// TIA Portal V18 export
// export: Created 2025-12-01T12:38:42.0092621Z, ExportSetting None, DisplayName Totally Integrated Automation Portal, DisplayVersion V18 Update 5, DisplayName TIA Portal Openness, DisplayVersion V18 Update 5, DisplayName TIA Portal Teamcenter Gateway, DisplayVersion V18, DisplayName TIA Portal Version Control Interface, DisplayVersion V18, DisplayName STEP 7 Professional, DisplayVersion V18 Update 5, DisplayName STEP 7 Safety, DisplayVersion V18, DisplayName WinCC Professional, DisplayVersion V18 Update 5
FUNCTION "Robot" : Void   // FC2400, LAD
{ S7_Optimized_Access := 'TRUE' }
// stored: AutoNumber false, SetENOAutomatically false
   VAR_TEMP   // added for the SCL form of the ladder/FBD networks
      _w1 : Bool;
      _w2 : Bool;
      _w3 : Bool;
      _w4 : Bool;
      _w5 : Bool;
      _w6 : Bool;
   END_VAR
BEGIN

REGION Network 1: 调用机器人1 / Call robot 1
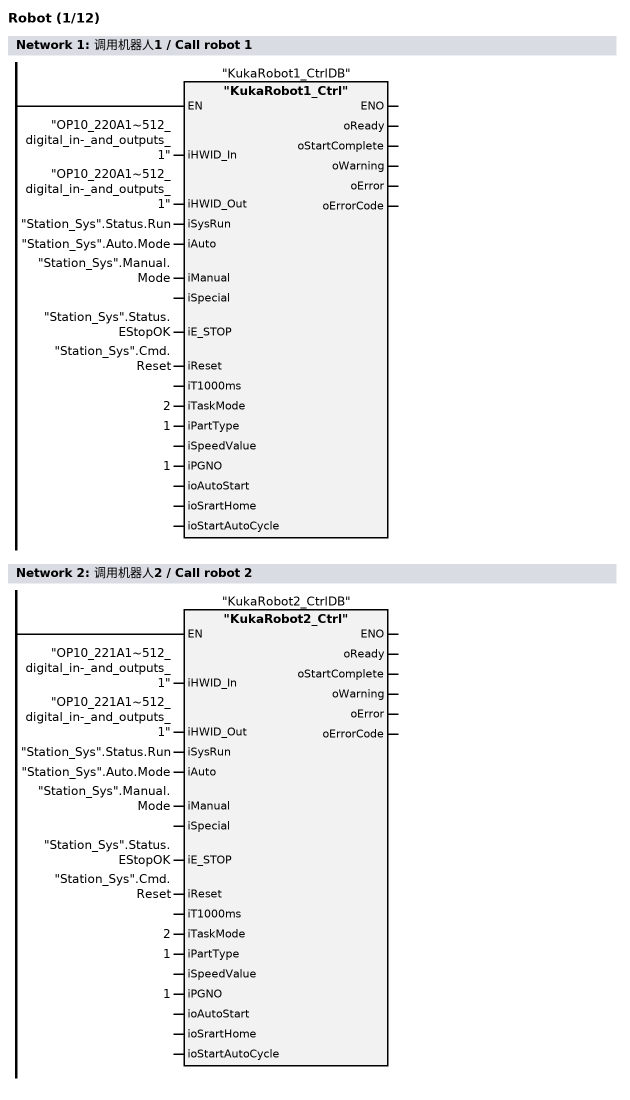
   RUNG wire#powerrail
      "KukaRobot1_CtrlDB"(iHWID_In := "OP10_220A1~512_digital_in-_and_outputs_1", iHWID_Out := "OP10_220A1~512_digital_in-_and_outputs_1", iSysRun := "Station_Sys".Status.Run, iAuto := "Station_Sys".Auto.Mode, iManual := "Station_Sys".Manual.Mode, iSpecial :=, iE_STOP := "Station_Sys".Status.EStopOK, iReset := "Station_Sys".Cmd.Reset, iT1000ms :=, iTaskMode := 2, iPartType := 1, iSpeedValue :=, iPGNO := 1, ioAutoStart :=, ioSrartHome :=, ioStartAutoCycle :=, oReady =>, oStartComplete =>, oWarning =>, oError =>, oErrorCode =>)
   END_RUNG
   // the same network as SCL:
   "KukaRobot1_CtrlDB"(iHWID_In := "OP10_220A1~512_digital_in-_and_outputs_1",   // "KukaRobot1_Ctrl"
                       iHWID_Out := "OP10_220A1~512_digital_in-_and_outputs_1",
                       iSysRun := "Station_Sys".Status.Run,
                       iAuto := "Station_Sys".Auto.Mode,
                       iManual := "Station_Sys".Manual.Mode,
                       iE_STOP := "Station_Sys".Status.EStopOK,
                       iReset := "Station_Sys".Cmd.Reset,
                       iTaskMode := 2,
                       iPartType := 1,
                       iPGNO := 1);
END_REGION

REGION Network 2: 调用机器人2 / Call robot 2
   RUNG wire#powerrail
      "KukaRobot2_CtrlDB"(iHWID_In := "OP10_221A1~512_digital_in-_and_outputs_1", iHWID_Out := "OP10_221A1~512_digital_in-_and_outputs_1", iSysRun := "Station_Sys".Status.Run, iAuto := "Station_Sys".Auto.Mode, iManual := "Station_Sys".Manual.Mode, iSpecial :=, iE_STOP := "Station_Sys".Status.EStopOK, iReset := "Station_Sys".Cmd.Reset, iT1000ms :=, iTaskMode := 2, iPartType := 1, iSpeedValue :=, iPGNO := 1, ioAutoStart :=, ioSrartHome :=, ioStartAutoCycle :=, oReady =>, oStartComplete =>, oWarning =>, oError =>, oErrorCode =>)
   END_RUNG
   // the same network as SCL:
   "KukaRobot2_CtrlDB"(iHWID_In := "OP10_221A1~512_digital_in-_and_outputs_1",   // "KukaRobot2_Ctrl"
                       iHWID_Out := "OP10_221A1~512_digital_in-_and_outputs_1",
                       iSysRun := "Station_Sys".Status.Run,
                       iAuto := "Station_Sys".Auto.Mode,
                       iManual := "Station_Sys".Manual.Mode,
                       iE_STOP := "Station_Sys".Status.EStopOK,
                       iReset := "Station_Sys".Cmd.Reset,
                       iTaskMode := 2,
                       iPartType := 1,
                       iPGNO := 1);
END_REGION

REGION Network 3: 调用机器人3 / Call robot 3
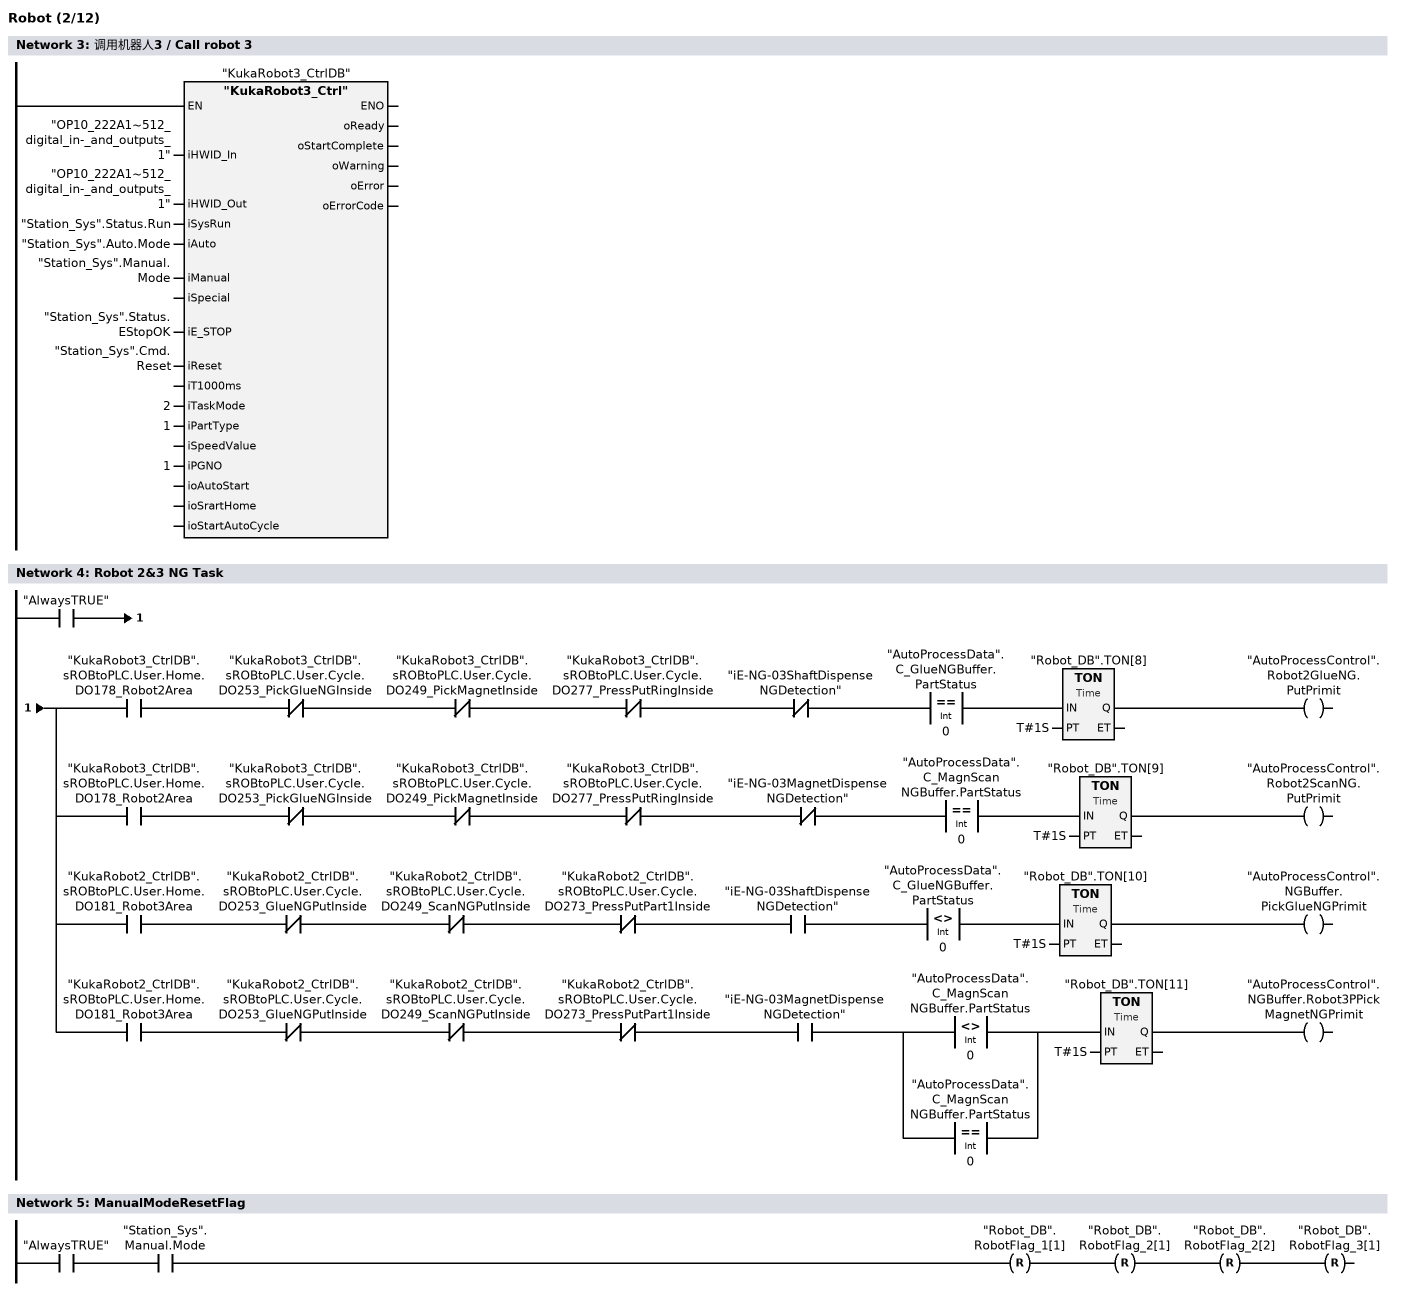
   RUNG wire#powerrail
      "KukaRobot3_CtrlDB"(iHWID_In := "OP10_222A1~512_digital_in-_and_outputs_1", iHWID_Out := "OP10_222A1~512_digital_in-_and_outputs_1", iSysRun := "Station_Sys".Status.Run, iAuto := "Station_Sys".Auto.Mode, iManual := "Station_Sys".Manual.Mode, iSpecial :=, iE_STOP := "Station_Sys".Status.EStopOK, iReset := "Station_Sys".Cmd.Reset, iT1000ms :=, iTaskMode := 2, iPartType := 1, iSpeedValue :=, iPGNO := 1, ioAutoStart :=, ioSrartHome :=, ioStartAutoCycle :=, oReady =>, oStartComplete =>, oWarning =>, oError =>, oErrorCode =>)
   END_RUNG
   // the same network as SCL:
   "KukaRobot3_CtrlDB"(iHWID_In := "OP10_222A1~512_digital_in-_and_outputs_1",   // "KukaRobot3_Ctrl"
                       iHWID_Out := "OP10_222A1~512_digital_in-_and_outputs_1",
                       iSysRun := "Station_Sys".Status.Run,
                       iAuto := "Station_Sys".Auto.Mode,
                       iManual := "Station_Sys".Manual.Mode,
                       iE_STOP := "Station_Sys".Status.EStopOK,
                       iReset := "Station_Sys".Cmd.Reset,
                       iTaskMode := 2,
                       iPartType := 1,
                       iPGNO := 1);
END_REGION

REGION Network 4: Robot 2&3 NG Task
   RUNG wire#powerrail
      Contact( "AlwaysTRUE" )
      wire#w1
      Contact( "KukaRobot3_CtrlDB".sROBtoPLC.User.Home.DO178_Robot2Area )
      I_Contact( "KukaRobot3_CtrlDB".sROBtoPLC.User.Cycle.DO253_PickGlueNGInside )
      I_Contact( "KukaRobot3_CtrlDB".sROBtoPLC.User.Cycle.DO249_PickMagnetInside )
      I_Contact( "KukaRobot3_CtrlDB".sROBtoPLC.User.Cycle.DO277_PressPutRingInside )
      I_Contact( "iE-NG-03ShaftDispenseNGDetection" )
      { S7_Templates := "SrcType := Int" } EQ_Contact(in1 := "AutoProcessData".C_GlueNGBuffer.PartStatus, in2 := 0)
      { S7_Templates := "time_type := Time" } "Robot_DB".TON[8].TON(pt := T#1S, et =>)
      Coil( "AutoProcessControl".Robot2GlueNG.PutPrimit )
   END_RUNG
   RUNG wire#w1
      Contact( "KukaRobot3_CtrlDB".sROBtoPLC.User.Home.DO178_Robot2Area )
      I_Contact( "KukaRobot3_CtrlDB".sROBtoPLC.User.Cycle.DO253_PickGlueNGInside )
      I_Contact( "KukaRobot3_CtrlDB".sROBtoPLC.User.Cycle.DO249_PickMagnetInside )
      I_Contact( "KukaRobot3_CtrlDB".sROBtoPLC.User.Cycle.DO277_PressPutRingInside )
      I_Contact( "iE-NG-03MagnetDispenseNGDetection" )
      { S7_Templates := "SrcType := Int" } EQ_Contact(in1 := "AutoProcessData".C_MagnScanNGBuffer.PartStatus, in2 := 0)
      { S7_Templates := "time_type := Time" } "Robot_DB".TON[9].TON(pt := T#1S, et =>)
      Coil( "AutoProcessControl".Robot2ScanNG.PutPrimit )
   END_RUNG
   RUNG wire#w1
      Contact( "KukaRobot2_CtrlDB".sROBtoPLC.User.Home.DO181_Robot3Area )
      I_Contact( "KukaRobot2_CtrlDB".sROBtoPLC.User.Cycle.DO253_GlueNGPutInside )
      I_Contact( "KukaRobot2_CtrlDB".sROBtoPLC.User.Cycle.DO249_ScanNGPutInside )
      I_Contact( "KukaRobot2_CtrlDB".sROBtoPLC.User.Cycle.DO273_PressPutPart1Inside )
      Contact( "iE-NG-03ShaftDispenseNGDetection" )
      { S7_Templates := "SrcType := Int" } NE_Contact(in1 := "AutoProcessData".C_GlueNGBuffer.PartStatus, in2 := 0)
      { S7_Templates := "time_type := Time" } "Robot_DB".TON[10].TON(pt := T#1S, et =>)
      Coil( "AutoProcessControl".NGBuffer.PickGlueNGPrimit )
   END_RUNG
   RUNG wire#w1
      Contact( "KukaRobot2_CtrlDB".sROBtoPLC.User.Home.DO181_Robot3Area )
      I_Contact( "KukaRobot2_CtrlDB".sROBtoPLC.User.Cycle.DO253_GlueNGPutInside )
      I_Contact( "KukaRobot2_CtrlDB".sROBtoPLC.User.Cycle.DO249_ScanNGPutInside )
      I_Contact( "KukaRobot2_CtrlDB".sROBtoPLC.User.Cycle.DO273_PressPutPart1Inside )
      Contact( "iE-NG-03MagnetDispenseNGDetection" )
      wire#w2
      { S7_Templates := "SrcType := Int" } NE_Contact(in1 := "AutoProcessData".C_MagnScanNGBuffer.PartStatus, in2 := 0)
      wire#w3
      { S7_Templates := "time_type := Time" } "Robot_DB".TON[11].TON(pt := T#1S, et =>)
      Coil( "AutoProcessControl".NGBuffer.Robot3PPickMagnetNGPrimit )
   END_RUNG
   RUNG wire#w2
      { S7_Templates := "SrcType := Int" } EQ_Contact(in1 := "AutoProcessData".C_MagnScanNGBuffer.PartStatus, in2 := 0)
   END_RUNG wire#w3
   // the same network as SCL:
   "Robot_DB".TON[8].TON(IN := "AlwaysTRUE" AND "KukaRobot3_CtrlDB".sROBtoPLC.User.Home.DO178_Robot2Area AND NOT "KukaRobot3_CtrlDB".sROBtoPLC.User.Cycle.DO253_PickGlueNGInside AND NOT "KukaRobot3_CtrlDB".sROBtoPLC.User.Cycle.DO249_PickMagnetInside AND NOT "KukaRobot3_CtrlDB".sROBtoPLC.User.Cycle.DO277_PressPutRingInside AND NOT "iE-NG-03ShaftDispenseNGDetection" AND ("AutoProcessData".C_GlueNGBuffer.PartStatus = 0),
                         PT := T#1S);
   "AutoProcessControl".Robot2GlueNG.PutPrimit := "Robot_DB".TON[8].Q;
   "Robot_DB".TON[9].TON(IN := "AlwaysTRUE" AND "KukaRobot3_CtrlDB".sROBtoPLC.User.Home.DO178_Robot2Area AND NOT "KukaRobot3_CtrlDB".sROBtoPLC.User.Cycle.DO253_PickGlueNGInside AND NOT "KukaRobot3_CtrlDB".sROBtoPLC.User.Cycle.DO249_PickMagnetInside AND NOT "KukaRobot3_CtrlDB".sROBtoPLC.User.Cycle.DO277_PressPutRingInside AND NOT "iE-NG-03MagnetDispenseNGDetection" AND ("AutoProcessData".C_MagnScanNGBuffer.PartStatus = 0),
                         PT := T#1S);
   "AutoProcessControl".Robot2ScanNG.PutPrimit := "Robot_DB".TON[9].Q;
   "Robot_DB".TON[10].TON(IN := "AlwaysTRUE" AND "KukaRobot2_CtrlDB".sROBtoPLC.User.Home.DO181_Robot3Area AND NOT "KukaRobot2_CtrlDB".sROBtoPLC.User.Cycle.DO253_GlueNGPutInside AND NOT "KukaRobot2_CtrlDB".sROBtoPLC.User.Cycle.DO249_ScanNGPutInside AND NOT "KukaRobot2_CtrlDB".sROBtoPLC.User.Cycle.DO273_PressPutPart1Inside AND "iE-NG-03ShaftDispenseNGDetection" AND ("AutoProcessData".C_GlueNGBuffer.PartStatus <> 0),
                          PT := T#1S);
   "AutoProcessControl".NGBuffer.PickGlueNGPrimit := "Robot_DB".TON[10].Q;
   "Robot_DB".TON[11].TON(IN := "AlwaysTRUE" AND "KukaRobot2_CtrlDB".sROBtoPLC.User.Home.DO181_Robot3Area AND NOT "KukaRobot2_CtrlDB".sROBtoPLC.User.Cycle.DO253_GlueNGPutInside AND NOT "KukaRobot2_CtrlDB".sROBtoPLC.User.Cycle.DO249_ScanNGPutInside AND NOT "KukaRobot2_CtrlDB".sROBtoPLC.User.Cycle.DO273_PressPutPart1Inside AND "iE-NG-03MagnetDispenseNGDetection" AND (("AutoProcessData".C_MagnScanNGBuffer.PartStatus <> 0) OR ("AutoProcessData".C_MagnScanNGBuffer.PartStatus = 0)),
                          PT := T#1S);
   "AutoProcessControl".NGBuffer.Robot3PPickMagnetNGPrimit := "Robot_DB".TON[11].Q;
END_REGION

REGION Network 5: ManualModeResetFlag
   RUNG wire#powerrail
      Contact( "AlwaysTRUE" )
      Contact( "Station_Sys".Manual.Mode )
      R_Coil( "Robot_DB".RobotFlag_1[1] )
      R_Coil( "Robot_DB".RobotFlag_2[1] )
      R_Coil( "Robot_DB".RobotFlag_2[2] )
      R_Coil( "Robot_DB".RobotFlag_3[1] )
   END_RUNG
   // the same network as SCL:
   IF "AlwaysTRUE" AND "Station_Sys".Manual.Mode THEN
       "Robot_DB".RobotFlag_1[1] := FALSE;
       "Robot_DB".RobotFlag_2[1] := FALSE;
       "Robot_DB".RobotFlag_2[2] := FALSE;
       "Robot_DB".RobotFlag_3[1] := FALSE;
   END_IF;
END_REGION

REGION Network 6 (SCL): LoadNG传感器 / Loadng sensor
   //NG1
   "KukaRobot1_CtrlDB".sPLCtoROB.User.Home.DI177_NG1_1:="Robot_DB".LoadNG_1[1] := "iE1-UnloadingShaftPressNG_5";
   "KukaRobot1_CtrlDB".sPLCtoROB.User.Home.DI178_NG1_2:="Robot_DB".LoadNG_1[2] := "iE1-UnloadingShaftPressNG_4";
   "KukaRobot1_CtrlDB".sPLCtoROB.User.Home.DI179_NG1_3:="Robot_DB".LoadNG_1[3] := "iE1-UnloadingShaftPressNG_3";
   "KukaRobot1_CtrlDB".sPLCtoROB.User.Home.DI180_NG1_4:="Robot_DB".LoadNG_1[4] := "iE1-UnloadingShaftPressNG_2";
   "KukaRobot1_CtrlDB".sPLCtoROB.User.Home.DI181_NG1_5:="Robot_DB".LoadNG_1[5] := "iE1-UnloadingShaftPressNG_1";

   //NG2
   "KukaRobot1_CtrlDB".sPLCtoROB.User.Home.DI182_NG2_1:="Robot_DB".LoadNG_2[1] := "iE1-UnloadingShaftScanNG_5";
   "KukaRobot1_CtrlDB".sPLCtoROB.User.Home.DI183_NG2_2:="Robot_DB".LoadNG_2[2] := "iE1-UnloadingShaftScanNG_4";
   "KukaRobot1_CtrlDB".sPLCtoROB.User.Home.DI184_NG2_3:="Robot_DB".LoadNG_2[3] := "iE1-UnloadingShaftScanNG_3";
   "KukaRobot1_CtrlDB".sPLCtoROB.User.Home.DI185_NG2_4:="Robot_DB".LoadNG_2[4] := "iE1-UnloadingShaftScanNG_2";
   "KukaRobot1_CtrlDB".sPLCtoROB.User.Home.DI186_NG2_5:="Robot_DB".LoadNG_2[5] := "iE1-UnloadingShaftScanNG_1";

   //NG3
   "KukaRobot1_CtrlDB".sPLCtoROB.User.Home.DI187_NG3_1:="Robot_DB".LoadNG_3[1] := "iE1-UnloadingRingScanNG_5";
   "KukaRobot1_CtrlDB".sPLCtoROB.User.Home.DI188_NG3_2:="Robot_DB".LoadNG_3[2] := "iE1-UnloadingRingScanNG_4";
   "KukaRobot1_CtrlDB".sPLCtoROB.User.Home.DI189_NG3_3:="Robot_DB".LoadNG_3[3] := "iE1-UnloadingRingScanNG_3";
   "KukaRobot1_CtrlDB".sPLCtoROB.User.Home.DI190_NG3_4:="Robot_DB".LoadNG_3[4] := "iE1-UnloadingRingScanNG_2";
   "KukaRobot1_CtrlDB".sPLCtoROB.User.Home.DI191_NG3_5:="Robot_DB".LoadNG_3[5] := "iE1-UnloadingRingScanNG_1";
END_REGION

REGION Network 7 (SCL): UnLoadNG传感器 / UnLoadNG sensor
   //NG1
   "KukaRobot3_CtrlDB".sPLCtoROB.User.Home.DI177_PressNG1_1:="Robot_DB".UnLoadNG_1[1] := "iE2-UnloadingPressNG_5";
   "KukaRobot3_CtrlDB".sPLCtoROB.User.Home.DI178_PressNG1_2:="Robot_DB".UnLoadNG_1[2] := "iE2-UnloadingPressNG_4";
   "KukaRobot3_CtrlDB".sPLCtoROB.User.Home.DI179_PressNG1_3:="Robot_DB".UnLoadNG_1[3] := "iE2-UnloadingPressNG_3";
   "KukaRobot3_CtrlDB".sPLCtoROB.User.Home.DI180_PressNG1_4:="Robot_DB".UnLoadNG_1[4] := "iE2-UnloadingPressNG_2";
   "KukaRobot3_CtrlDB".sPLCtoROB.User.Home.DI181_PressNG1_5:="Robot_DB".UnLoadNG_1[5] := "iE2-UnloadingPressNG_1";

   //NG2
   "KukaRobot3_CtrlDB".sPLCtoROB.User.Home.DI182_GlueNG2_1:="Robot_DB".UnLoadNG_2[1] := "iE2-UnloadingMagentScanNG_5";
   "KukaRobot3_CtrlDB".sPLCtoROB.User.Home.DI183_GlueNG2_2:="Robot_DB".UnLoadNG_2[2] := "iE2-UnloadingMagentScanNG_4";
   "KukaRobot3_CtrlDB".sPLCtoROB.User.Home.DI184_GlueNG2_3:="Robot_DB".UnLoadNG_2[3] := "iE2-UnloadingMagentScanNG_3";
   "KukaRobot3_CtrlDB".sPLCtoROB.User.Home.DI185_GlueNG2_4:="Robot_DB".UnLoadNG_2[4] := "iE2-UnloadingMagentScanNG_2";
   "KukaRobot3_CtrlDB".sPLCtoROB.User.Home.DI186_GlueNG2_5:="Robot_DB".UnLoadNG_2[5] := "iE2-UnloadingMagentScanNG_1";

   //NG3
   "KukaRobot3_CtrlDB".sPLCtoROB.User.Home.DI187_ScanNG3_1:="Robot_DB".UnLoadNG_3[1] := "iE2-UnloadingRingScanNG_5";
   "KukaRobot3_CtrlDB".sPLCtoROB.User.Home.DI188_ScanNG3_2:="Robot_DB".UnLoadNG_3[2] := "iE2-UnloadingRingScanNG_4";
   "KukaRobot3_CtrlDB".sPLCtoROB.User.Home.DI189_ScanNG3_3:="Robot_DB".UnLoadNG_3[3] := "iE2-UnloadingRingScanNG_3";
   "KukaRobot3_CtrlDB".sPLCtoROB.User.Home.DI190_ScanNG3_4:="Robot_DB".UnLoadNG_3[4] := "iE2-UnloadingRingScanNG_2";
   "KukaRobot3_CtrlDB".sPLCtoROB.User.Home.DI191_ScanNG3_5:="Robot_DB".UnLoadNG_3[5] := "iE2-UnloadingRingScanNG_1";
END_REGION

REGION Network 8: RobotGripControl
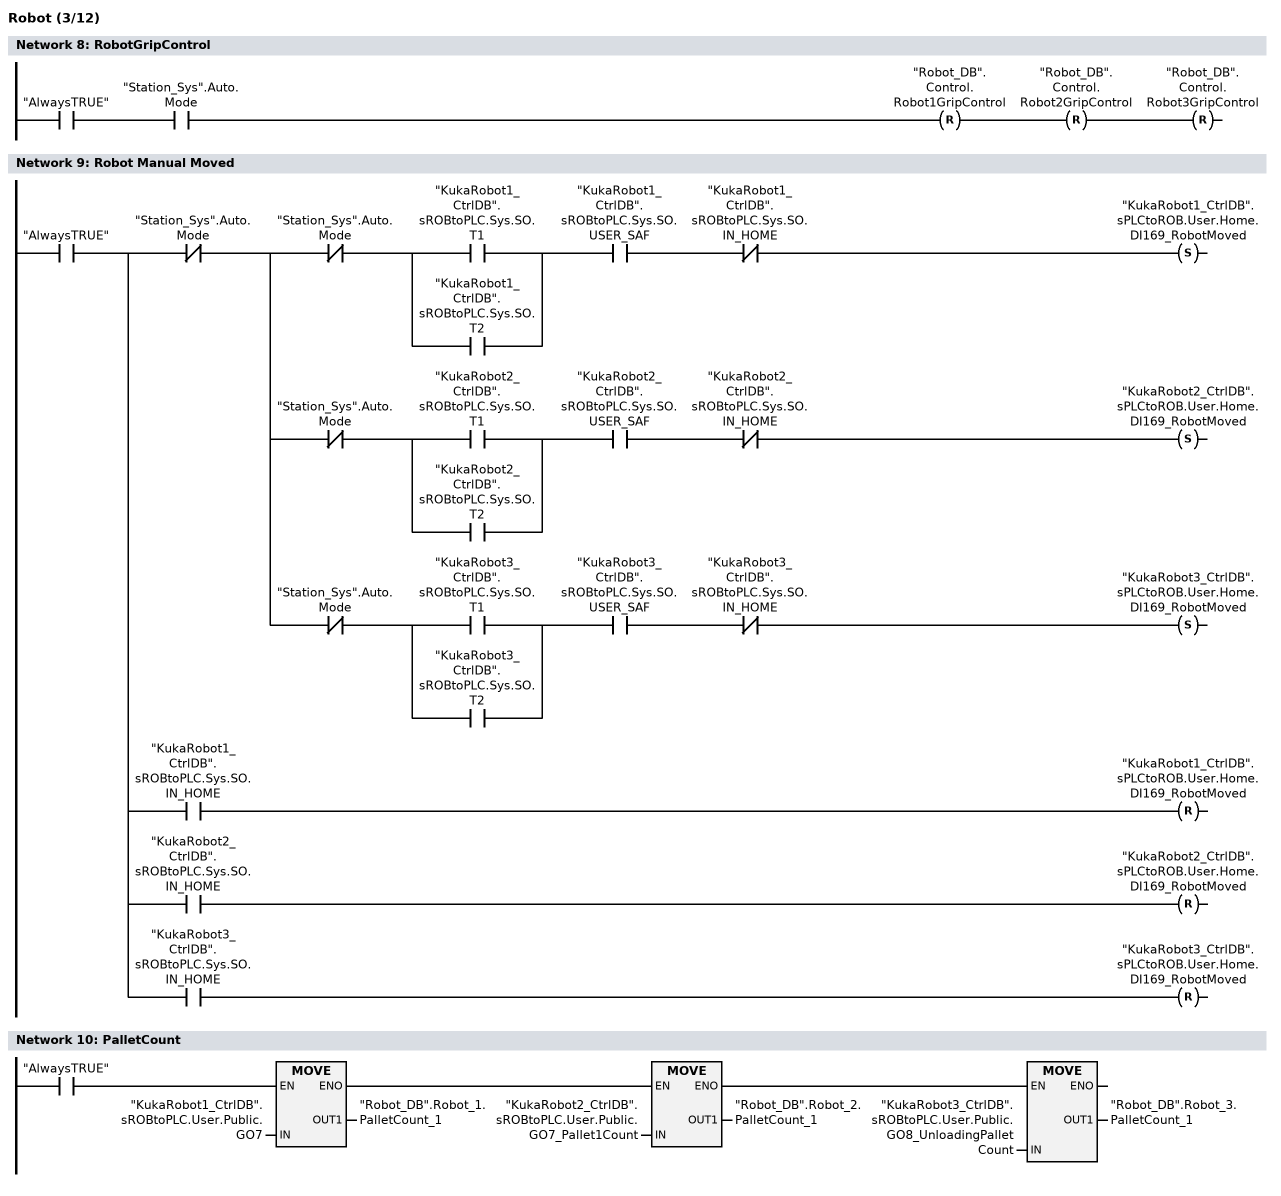
   RUNG wire#powerrail
      Contact( "AlwaysTRUE" )
      Contact( "Station_Sys".Auto.Mode )
      R_Coil( "Robot_DB".Control.Robot1GripControl )
      R_Coil( "Robot_DB".Control.Robot2GripControl )
      R_Coil( "Robot_DB".Control.Robot3GripControl )
   END_RUNG
   // the same network as SCL:
   IF "AlwaysTRUE" AND "Station_Sys".Auto.Mode THEN
       "Robot_DB".Control.Robot1GripControl := FALSE;
       "Robot_DB".Control.Robot2GripControl := FALSE;
       "Robot_DB".Control.Robot3GripControl := FALSE;
   END_IF;
END_REGION

REGION Network 9: Robot Manual Moved
   RUNG wire#powerrail
      Contact( "AlwaysTRUE" )
      wire#w1
      I_Contact( "Station_Sys".Auto.Mode )
      wire#w2
      I_Contact( "Station_Sys".Auto.Mode )
      wire#w3
      Contact( "KukaRobot1_CtrlDB".sROBtoPLC.Sys.SO.T1 )
      wire#w4
      Contact( "KukaRobot1_CtrlDB".sROBtoPLC.Sys.SO.USER_SAF )
      I_Contact( "KukaRobot1_CtrlDB".sROBtoPLC.Sys.SO.IN_HOME )
      S_Coil( "KukaRobot1_CtrlDB".sPLCtoROB.User.Home.DI169_RobotMoved )
   END_RUNG
   RUNG wire#w3
      Contact( "KukaRobot1_CtrlDB".sROBtoPLC.Sys.SO.T2 )
   END_RUNG wire#w4
   RUNG wire#w2
      I_Contact( "Station_Sys".Auto.Mode )
      wire#w5
      Contact( "KukaRobot2_CtrlDB".sROBtoPLC.Sys.SO.T1 )
      wire#w6
      Contact( "KukaRobot2_CtrlDB".sROBtoPLC.Sys.SO.USER_SAF )
      I_Contact( "KukaRobot2_CtrlDB".sROBtoPLC.Sys.SO.IN_HOME )
      S_Coil( "KukaRobot2_CtrlDB".sPLCtoROB.User.Home.DI169_RobotMoved )
   END_RUNG
   RUNG wire#w5
      Contact( "KukaRobot2_CtrlDB".sROBtoPLC.Sys.SO.T2 )
   END_RUNG wire#w6
   RUNG wire#w2
      I_Contact( "Station_Sys".Auto.Mode )
      wire#w7
      Contact( "KukaRobot3_CtrlDB".sROBtoPLC.Sys.SO.T1 )
      wire#w8
      Contact( "KukaRobot3_CtrlDB".sROBtoPLC.Sys.SO.USER_SAF )
      I_Contact( "KukaRobot3_CtrlDB".sROBtoPLC.Sys.SO.IN_HOME )
      S_Coil( "KukaRobot3_CtrlDB".sPLCtoROB.User.Home.DI169_RobotMoved )
   END_RUNG
   RUNG wire#w7
      Contact( "KukaRobot3_CtrlDB".sROBtoPLC.Sys.SO.T2 )
   END_RUNG wire#w8
   RUNG wire#w1
      Contact( "KukaRobot1_CtrlDB".sROBtoPLC.Sys.SO.IN_HOME )
      R_Coil( "KukaRobot1_CtrlDB".sPLCtoROB.User.Home.DI169_RobotMoved )
   END_RUNG
   RUNG wire#w1
      Contact( "KukaRobot2_CtrlDB".sROBtoPLC.Sys.SO.IN_HOME )
      R_Coil( "KukaRobot2_CtrlDB".sPLCtoROB.User.Home.DI169_RobotMoved )
   END_RUNG
   RUNG wire#w1
      Contact( "KukaRobot3_CtrlDB".sROBtoPLC.Sys.SO.IN_HOME )
      R_Coil( "KukaRobot3_CtrlDB".sPLCtoROB.User.Home.DI169_RobotMoved )
   END_RUNG
   // the same network as SCL:
   #_w1 := "AlwaysTRUE" AND NOT "Station_Sys".Auto.Mode;
   IF #_w1 AND NOT "Station_Sys".Auto.Mode AND ("KukaRobot1_CtrlDB".sROBtoPLC.Sys.SO.T1 OR "KukaRobot1_CtrlDB".sROBtoPLC.Sys.SO.T2) AND "KukaRobot1_CtrlDB".sROBtoPLC.Sys.SO.USER_SAF AND NOT "KukaRobot1_CtrlDB".sROBtoPLC.Sys.SO.IN_HOME THEN
       "KukaRobot1_CtrlDB".sPLCtoROB.User.Home.DI169_RobotMoved := TRUE;
   END_IF;
   IF #_w1 AND NOT "Station_Sys".Auto.Mode AND ("KukaRobot2_CtrlDB".sROBtoPLC.Sys.SO.T1 OR "KukaRobot2_CtrlDB".sROBtoPLC.Sys.SO.T2) AND "KukaRobot2_CtrlDB".sROBtoPLC.Sys.SO.USER_SAF AND NOT "KukaRobot2_CtrlDB".sROBtoPLC.Sys.SO.IN_HOME THEN
       "KukaRobot2_CtrlDB".sPLCtoROB.User.Home.DI169_RobotMoved := TRUE;
   END_IF;
   IF #_w1 AND NOT "Station_Sys".Auto.Mode AND ("KukaRobot3_CtrlDB".sROBtoPLC.Sys.SO.T1 OR "KukaRobot3_CtrlDB".sROBtoPLC.Sys.SO.T2) AND "KukaRobot3_CtrlDB".sROBtoPLC.Sys.SO.USER_SAF AND NOT "KukaRobot3_CtrlDB".sROBtoPLC.Sys.SO.IN_HOME THEN
       "KukaRobot3_CtrlDB".sPLCtoROB.User.Home.DI169_RobotMoved := TRUE;
   END_IF;
   IF "AlwaysTRUE" AND "KukaRobot1_CtrlDB".sROBtoPLC.Sys.SO.IN_HOME THEN
       "KukaRobot1_CtrlDB".sPLCtoROB.User.Home.DI169_RobotMoved := FALSE;
   END_IF;
   IF "AlwaysTRUE" AND "KukaRobot2_CtrlDB".sROBtoPLC.Sys.SO.IN_HOME THEN
       "KukaRobot2_CtrlDB".sPLCtoROB.User.Home.DI169_RobotMoved := FALSE;
   END_IF;
   IF "AlwaysTRUE" AND "KukaRobot3_CtrlDB".sROBtoPLC.Sys.SO.IN_HOME THEN
       "KukaRobot3_CtrlDB".sPLCtoROB.User.Home.DI169_RobotMoved := FALSE;
   END_IF;
END_REGION

REGION Network 10: PalletCount
   RUNG wire#powerrail
      Contact( "AlwaysTRUE" )
      Move(in := "KukaRobot1_CtrlDB".sROBtoPLC.User.Public.GO7, out1 => "Robot_DB".Robot_1.PalletCount_1)
      Move(in := "KukaRobot2_CtrlDB".sROBtoPLC.User.Public.GO7_Pallet1Count, out1 => "Robot_DB".Robot_2.PalletCount_1)
      Move(in := "KukaRobot3_CtrlDB".sROBtoPLC.User.Public.GO8_UnloadingPalletCount, out1 => "Robot_DB".Robot_3.PalletCount_1)
   END_RUNG
   // the same network as SCL:
   IF "AlwaysTRUE" THEN
       "Robot_DB".Robot_1.PalletCount_1 := "KukaRobot1_CtrlDB".sROBtoPLC.User.Public.GO7;
       "Robot_DB".Robot_2.PalletCount_1 := "KukaRobot2_CtrlDB".sROBtoPLC.User.Public.GO7_Pallet1Count;
       "Robot_DB".Robot_3.PalletCount_1 := "KukaRobot3_CtrlDB".sROBtoPLC.User.Public.GO8_UnloadingPalletCount;
   END_IF;
END_REGION

REGION Network 12: ----------------------------------------- Robot_1 -------------------------------------
END_REGION

REGION Network 13: CodeCompare
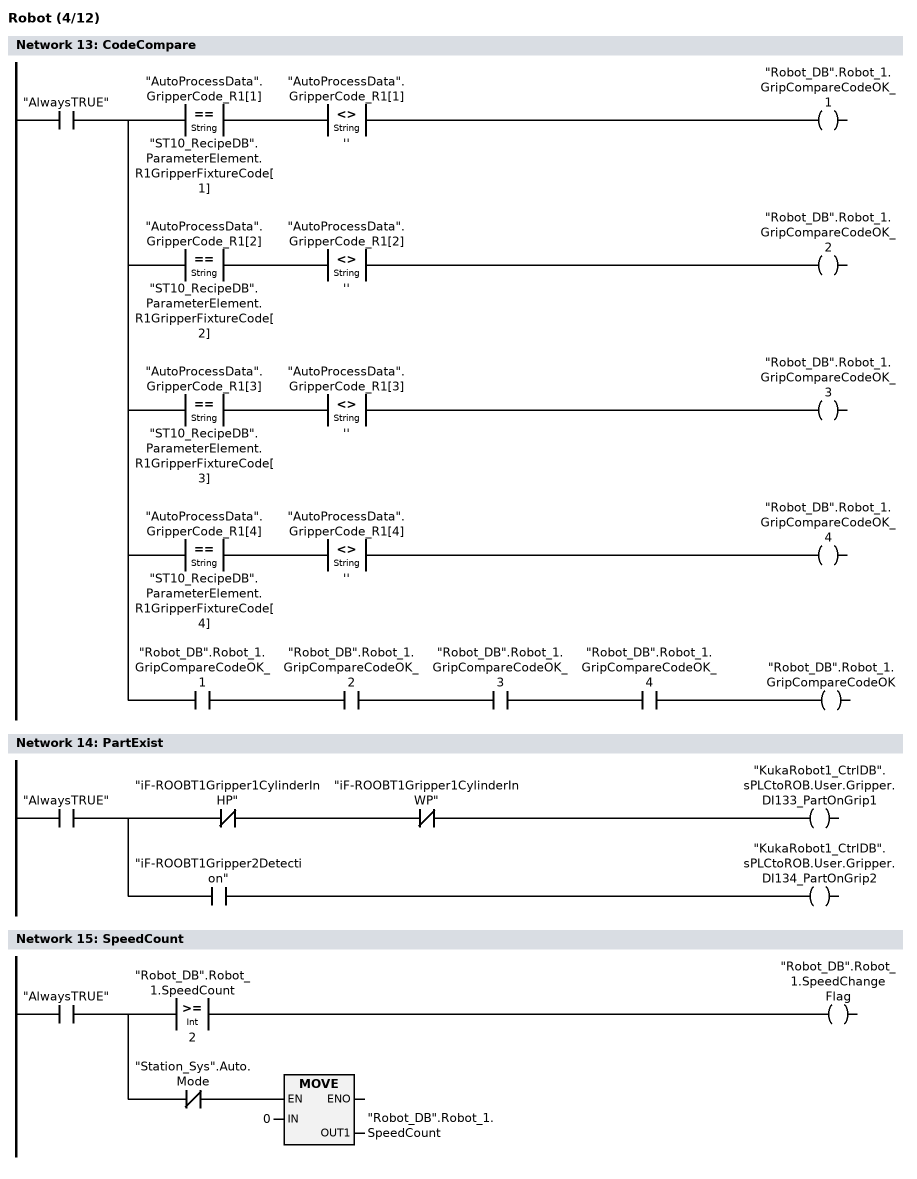
   RUNG wire#powerrail
      Contact( "AlwaysTRUE" )
      wire#w1
      { S7_Templates := "SrcType := String" } EQ_Contact(in1 := "AutoProcessData".GripperCode_R1[1], in2 := "ST10_RecipeDB".ParameterElement.R1GripperFixtureCode[1])
      { S7_Templates := "SrcType := String" } NE_Contact(in1 := "AutoProcessData".GripperCode_R1[1], in2 := '')
      Coil( "Robot_DB".Robot_1.GripCompareCodeOK_1 )
   END_RUNG
   RUNG wire#w1
      { S7_Templates := "SrcType := String" } EQ_Contact(in1 := "AutoProcessData".GripperCode_R1[2], in2 := "ST10_RecipeDB".ParameterElement.R1GripperFixtureCode[2])
      { S7_Templates := "SrcType := String" } NE_Contact(in1 := "AutoProcessData".GripperCode_R1[2], in2 := '')
      Coil( "Robot_DB".Robot_1.GripCompareCodeOK_2 )
   END_RUNG
   RUNG wire#w1
      { S7_Templates := "SrcType := String" } EQ_Contact(in1 := "AutoProcessData".GripperCode_R1[3], in2 := "ST10_RecipeDB".ParameterElement.R1GripperFixtureCode[3])
      { S7_Templates := "SrcType := String" } NE_Contact(in1 := "AutoProcessData".GripperCode_R1[3], in2 := '')
      Coil( "Robot_DB".Robot_1.GripCompareCodeOK_3 )
   END_RUNG
   RUNG wire#w1
      { S7_Templates := "SrcType := String" } EQ_Contact(in1 := "AutoProcessData".GripperCode_R1[4], in2 := "ST10_RecipeDB".ParameterElement.R1GripperFixtureCode[4])
      { S7_Templates := "SrcType := String" } NE_Contact(in1 := "AutoProcessData".GripperCode_R1[4], in2 := '')
      Coil( "Robot_DB".Robot_1.GripCompareCodeOK_4 )
   END_RUNG
   RUNG wire#w1
      Contact( "Robot_DB".Robot_1.GripCompareCodeOK_1 )
      Contact( "Robot_DB".Robot_1.GripCompareCodeOK_2 )
      Contact( "Robot_DB".Robot_1.GripCompareCodeOK_3 )
      Contact( "Robot_DB".Robot_1.GripCompareCodeOK_4 )
      Coil( "Robot_DB".Robot_1.GripCompareCodeOK )
   END_RUNG
   // the same network as SCL:
   "Robot_DB".Robot_1.GripCompareCodeOK_1 := "AlwaysTRUE" AND ("AutoProcessData".GripperCode_R1[1] = "ST10_RecipeDB".ParameterElement.R1GripperFixtureCode[1]) AND ("AutoProcessData".GripperCode_R1[1] <> '');
   "Robot_DB".Robot_1.GripCompareCodeOK_2 := "AlwaysTRUE" AND ("AutoProcessData".GripperCode_R1[2] = "ST10_RecipeDB".ParameterElement.R1GripperFixtureCode[2]) AND ("AutoProcessData".GripperCode_R1[2] <> '');
   "Robot_DB".Robot_1.GripCompareCodeOK_3 := "AlwaysTRUE" AND ("AutoProcessData".GripperCode_R1[3] = "ST10_RecipeDB".ParameterElement.R1GripperFixtureCode[3]) AND ("AutoProcessData".GripperCode_R1[3] <> '');
   "Robot_DB".Robot_1.GripCompareCodeOK_4 := "AlwaysTRUE" AND ("AutoProcessData".GripperCode_R1[4] = "ST10_RecipeDB".ParameterElement.R1GripperFixtureCode[4]) AND ("AutoProcessData".GripperCode_R1[4] <> '');
   "Robot_DB".Robot_1.GripCompareCodeOK := "AlwaysTRUE" AND "Robot_DB".Robot_1.GripCompareCodeOK_1 AND "Robot_DB".Robot_1.GripCompareCodeOK_2 AND "Robot_DB".Robot_1.GripCompareCodeOK_3 AND "Robot_DB".Robot_1.GripCompareCodeOK_4;
END_REGION

REGION Network 14: PartExist
   RUNG wire#powerrail
      Contact( "AlwaysTRUE" )
      wire#w1
      I_Contact( "iF-ROOBT1Gripper1CylinderInHP" )
      I_Contact( "iF-ROOBT1Gripper1CylinderInWP" )
      Coil( "KukaRobot1_CtrlDB".sPLCtoROB.User.Gripper.DI133_PartOnGrip1 )
   END_RUNG
   RUNG wire#w1
      Contact( "iF-ROOBT1Gripper2Detection" )
      Coil( "KukaRobot1_CtrlDB".sPLCtoROB.User.Gripper.DI134_PartOnGrip2 )
   END_RUNG
   // the same network as SCL:
   "KukaRobot1_CtrlDB".sPLCtoROB.User.Gripper.DI133_PartOnGrip1 := "AlwaysTRUE" AND NOT "iF-ROOBT1Gripper1CylinderInHP" AND NOT "iF-ROOBT1Gripper1CylinderInWP";
   "KukaRobot1_CtrlDB".sPLCtoROB.User.Gripper.DI134_PartOnGrip2 := "AlwaysTRUE" AND "iF-ROOBT1Gripper2Detection";
END_REGION

REGION Network 15: SpeedCount
   RUNG wire#powerrail
      Contact( "AlwaysTRUE" )
      wire#w1
      { S7_Templates := "SrcType := Int" } GE_Contact(in1 := "Robot_DB".Robot_1.SpeedCount, in2 := 2)
      Coil( "Robot_DB".Robot_1.SpeedChangeFlag )
   END_RUNG
   RUNG wire#w1
      I_Contact( "Station_Sys".Auto.Mode )
      Move(in := 0, out1 => "Robot_DB".Robot_1.SpeedCount)
   END_RUNG
   // the same network as SCL:
   "Robot_DB".Robot_1.SpeedChangeFlag := "AlwaysTRUE" AND ("Robot_DB".Robot_1.SpeedCount >= 2);
   IF "AlwaysTRUE" AND NOT "Station_Sys".Auto.Mode THEN "Robot_DB".Robot_1.SpeedCount := 0; END_IF;
END_REGION

REGION Network 16: Robot1Speed Interlock
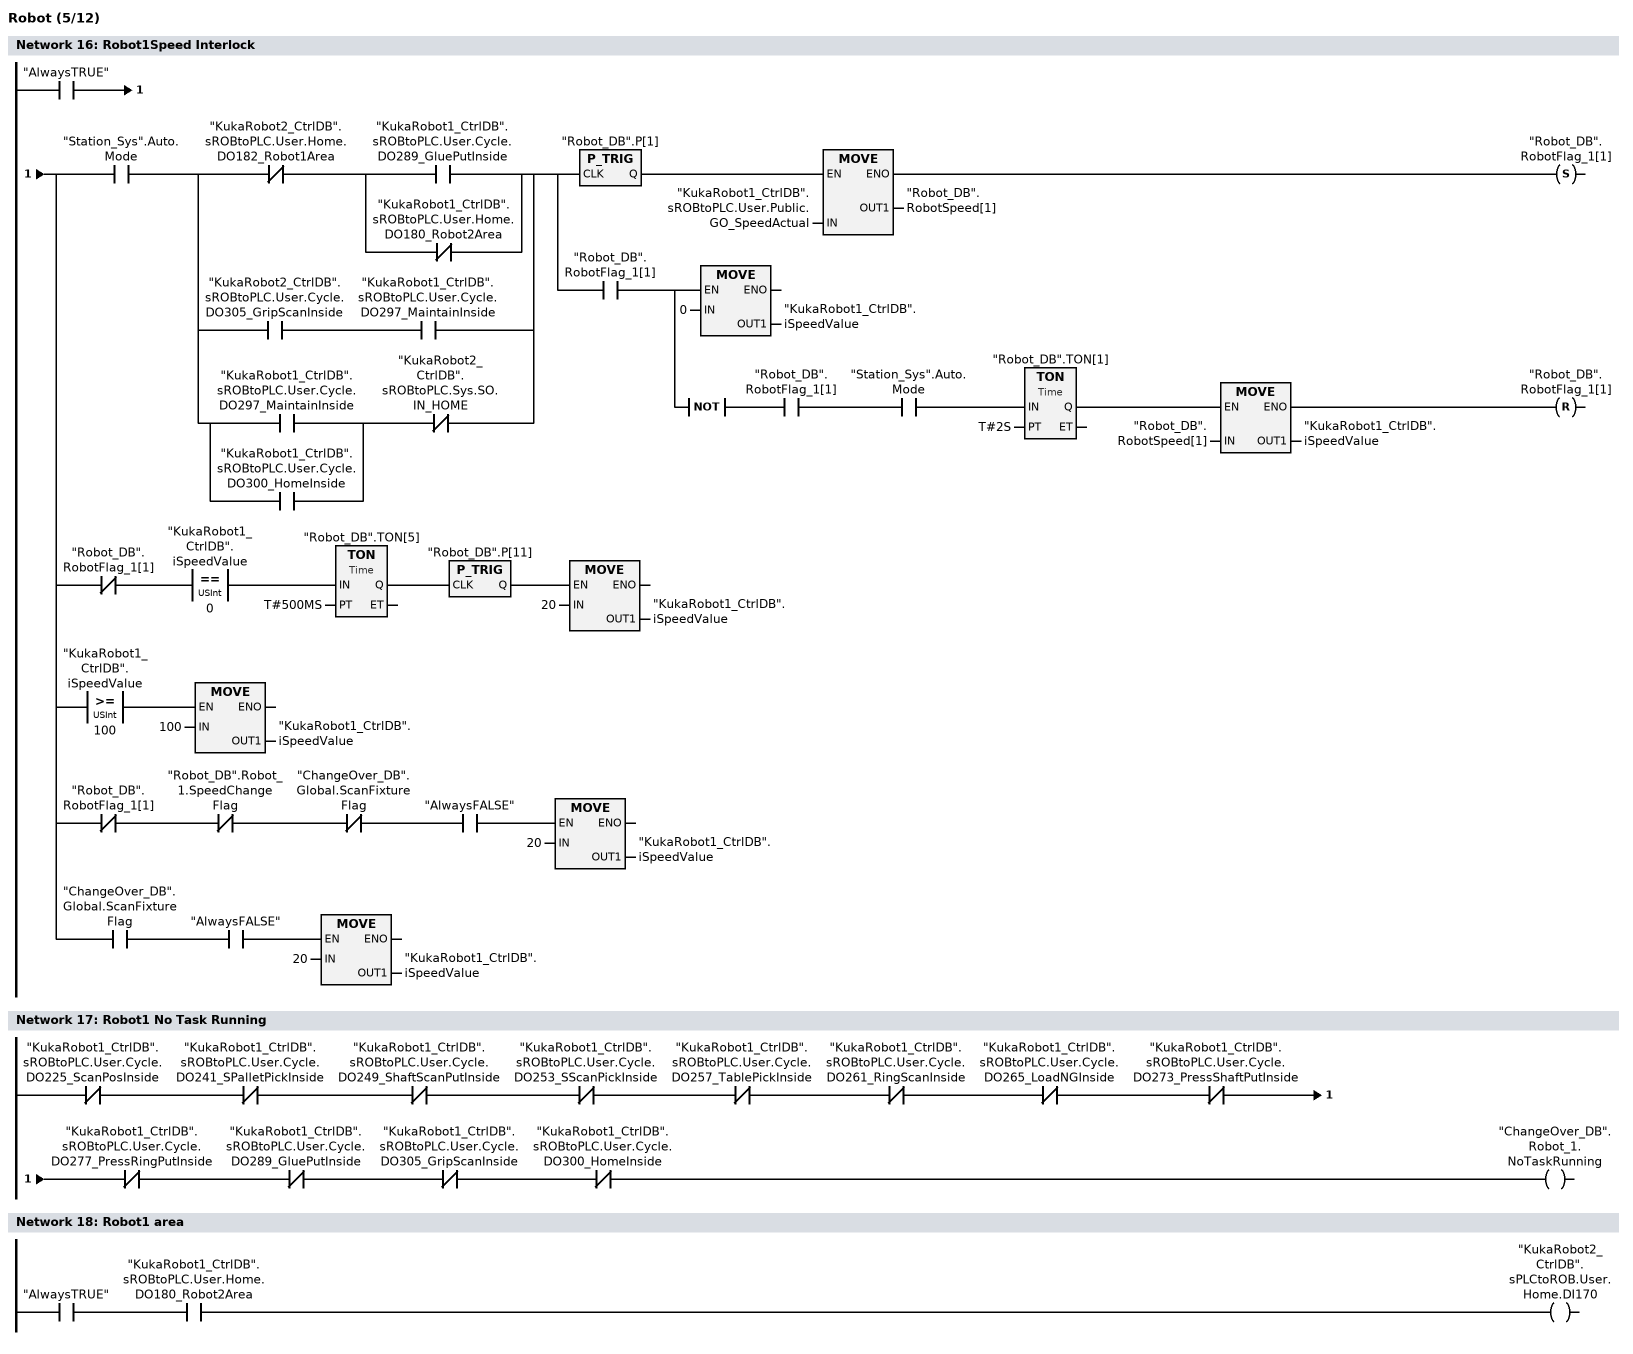
   RUNG wire#powerrail
      Contact( "AlwaysTRUE" )
      wire#w1
      Contact( "Station_Sys".Auto.Mode )
      wire#w2
      I_Contact( "KukaRobot2_CtrlDB".sROBtoPLC.User.Home.DO182_Robot1Area )
      wire#w3
      Contact( "KukaRobot1_CtrlDB".sROBtoPLC.User.Cycle.DO289_GluePutInside )
      wire#w4
      P_Trig( "Robot_DB".P[1] )
      Move(in := "KukaRobot1_CtrlDB".sROBtoPLC.User.Public.GO_SpeedActual, out1 => "Robot_DB".RobotSpeed[1])
      S_Coil( "Robot_DB".RobotFlag_1[1] )
   END_RUNG
   RUNG wire#w3
      I_Contact( "KukaRobot1_CtrlDB".sROBtoPLC.User.Home.DO180_Robot2Area )
   END_RUNG wire#w4
   RUNG wire#w2
      Contact( "KukaRobot2_CtrlDB".sROBtoPLC.User.Cycle.DO305_GripScanInside )
      Contact( "KukaRobot1_CtrlDB".sROBtoPLC.User.Cycle.DO297_MaintainInside )
   END_RUNG wire#w4
   RUNG wire#w2
      Contact( "KukaRobot1_CtrlDB".sROBtoPLC.User.Cycle.DO297_MaintainInside )
      wire#w5
      I_Contact( "KukaRobot2_CtrlDB".sROBtoPLC.Sys.SO.IN_HOME )
   END_RUNG wire#w4
   RUNG wire#w2
      Contact( "KukaRobot1_CtrlDB".sROBtoPLC.User.Cycle.DO300_HomeInside )
   END_RUNG wire#w5
   RUNG wire#w4
      Contact( "Robot_DB".RobotFlag_1[1] )
      wire#w6
      Move(in := 0, out1 => "KukaRobot1_CtrlDB".iSpeedValue)
   END_RUNG
   RUNG wire#w6
      Not()
      Contact( "Robot_DB".RobotFlag_1[1] )
      Contact( "Station_Sys".Auto.Mode )
      { S7_Templates := "time_type := Time" } "Robot_DB".TON[1].TON(pt := T#2S, et =>)
      Move(in := "Robot_DB".RobotSpeed[1], out1 => "KukaRobot1_CtrlDB".iSpeedValue)
      R_Coil( "Robot_DB".RobotFlag_1[1] )
   END_RUNG
   RUNG wire#w1
      I_Contact( "Robot_DB".RobotFlag_1[1] )
      { S7_Templates := "SrcType := USInt" } EQ_Contact(in1 := "KukaRobot1_CtrlDB".iSpeedValue, in2 := 0)
      { S7_Templates := "time_type := Time" } "Robot_DB".TON[5].TON(pt := T#500MS, et =>)
      P_Trig( "Robot_DB".P[11] )
      Move(in := 20, out1 => "KukaRobot1_CtrlDB".iSpeedValue)
   END_RUNG
   RUNG wire#w1
      { S7_Templates := "SrcType := USInt" } GE_Contact(in1 := "KukaRobot1_CtrlDB".iSpeedValue, in2 := 100)
      Move(in := 100, out1 => "KukaRobot1_CtrlDB".iSpeedValue)
   END_RUNG
   RUNG wire#w1
      I_Contact( "Robot_DB".RobotFlag_1[1] )
      I_Contact( "Robot_DB".Robot_1.SpeedChangeFlag )
      I_Contact( "ChangeOver_DB".Global.ScanFixtureFlag )
      Contact( "AlwaysFALSE" )
      Move(in := 20, out1 => "KukaRobot1_CtrlDB".iSpeedValue)
   END_RUNG
   RUNG wire#w1
      Contact( "ChangeOver_DB".Global.ScanFixtureFlag )
      Contact( "AlwaysFALSE" )
      Move(in := 20, out1 => "KukaRobot1_CtrlDB".iSpeedValue)
   END_RUNG
   // the same network as SCL:
   #_w1 := "AlwaysTRUE" AND "Station_Sys".Auto.Mode AND ((NOT "KukaRobot2_CtrlDB".sROBtoPLC.User.Home.DO182_Robot1Area AND ("KukaRobot1_CtrlDB".sROBtoPLC.User.Cycle.DO289_GluePutInside OR NOT "KukaRobot1_CtrlDB".sROBtoPLC.User.Home.DO180_Robot2Area)) OR ("KukaRobot2_CtrlDB".sROBtoPLC.User.Cycle.DO305_GripScanInside AND "KukaRobot1_CtrlDB".sROBtoPLC.User.Cycle.DO297_MaintainInside) OR (("KukaRobot1_CtrlDB".sROBtoPLC.User.Cycle.DO297_MaintainInside OR "KukaRobot1_CtrlDB".sROBtoPLC.User.Cycle.DO300_HomeInside) AND NOT "KukaRobot2_CtrlDB".sROBtoPLC.Sys.SO.IN_HOME));
   #_w2 := #_w1 AND NOT "Robot_DB".P[1];   // rising edge
   "Robot_DB".P[1] := #_w1;
   IF #_w2 THEN
       "Robot_DB".RobotSpeed[1] := "KukaRobot1_CtrlDB".sROBtoPLC.User.Public.GO_SpeedActual;
       "Robot_DB".RobotFlag_1[1] := TRUE;
   END_IF;
   #_w3 := #_w1 AND "Robot_DB".RobotFlag_1[1];
   IF #_w3 THEN "KukaRobot1_CtrlDB".iSpeedValue := 0; END_IF;
   "Robot_DB".TON[1].TON(IN := NOT #_w3 AND "Robot_DB".RobotFlag_1[1] AND "Station_Sys".Auto.Mode, PT := T#2S);
   IF "Robot_DB".TON[1].Q THEN
       "KukaRobot1_CtrlDB".iSpeedValue := "Robot_DB".RobotSpeed[1];
       "Robot_DB".RobotFlag_1[1] := FALSE;
   END_IF;
   "Robot_DB".TON[5].TON(IN := "AlwaysTRUE" AND NOT "Robot_DB".RobotFlag_1[1] AND ("KukaRobot1_CtrlDB".iSpeedValue = 0),
                         PT := T#500MS);
   #_w4 := "Robot_DB".TON[5].Q AND NOT "Robot_DB".P[11];   // rising edge
   "Robot_DB".P[11] := "Robot_DB".TON[5].Q;
   IF #_w4 THEN "KukaRobot1_CtrlDB".iSpeedValue := 20; END_IF;
   IF "AlwaysTRUE" AND ("KukaRobot1_CtrlDB".iSpeedValue >= 100) THEN
       "KukaRobot1_CtrlDB".iSpeedValue := 100;
   END_IF;
   IF "AlwaysTRUE" AND NOT "Robot_DB".RobotFlag_1[1] AND NOT "Robot_DB".Robot_1.SpeedChangeFlag AND NOT "ChangeOver_DB".Global.ScanFixtureFlag AND "AlwaysFALSE" THEN
       "KukaRobot1_CtrlDB".iSpeedValue := 20;
   END_IF;
   IF "AlwaysTRUE" AND "ChangeOver_DB".Global.ScanFixtureFlag AND "AlwaysFALSE" THEN
       "KukaRobot1_CtrlDB".iSpeedValue := 20;
   END_IF;
END_REGION

REGION Network 17: Robot1 No Task Running
   RUNG wire#powerrail
      I_Contact( "KukaRobot1_CtrlDB".sROBtoPLC.User.Cycle.DO225_ScanPosInside )
      I_Contact( "KukaRobot1_CtrlDB".sROBtoPLC.User.Cycle.DO241_SPalletPickInside )
      I_Contact( "KukaRobot1_CtrlDB".sROBtoPLC.User.Cycle.DO249_ShaftScanPutInside )
      I_Contact( "KukaRobot1_CtrlDB".sROBtoPLC.User.Cycle.DO253_SScanPickInside )
      I_Contact( "KukaRobot1_CtrlDB".sROBtoPLC.User.Cycle.DO257_TablePickInside )
      I_Contact( "KukaRobot1_CtrlDB".sROBtoPLC.User.Cycle.DO261_RingScanInside )
      I_Contact( "KukaRobot1_CtrlDB".sROBtoPLC.User.Cycle.DO265_LoadNGInside )
      I_Contact( "KukaRobot1_CtrlDB".sROBtoPLC.User.Cycle.DO273_PressShaftPutInside )
      I_Contact( "KukaRobot1_CtrlDB".sROBtoPLC.User.Cycle.DO277_PressRingPutInside )
      I_Contact( "KukaRobot1_CtrlDB".sROBtoPLC.User.Cycle.DO289_GluePutInside )
      I_Contact( "KukaRobot1_CtrlDB".sROBtoPLC.User.Cycle.DO305_GripScanInside )
      I_Contact( "KukaRobot1_CtrlDB".sROBtoPLC.User.Cycle.DO300_HomeInside )
      Coil( "ChangeOver_DB".Robot_1.NoTaskRunning )
   END_RUNG
   // the same network as SCL:
   "ChangeOver_DB".Robot_1.NoTaskRunning := NOT "KukaRobot1_CtrlDB".sROBtoPLC.User.Cycle.DO225_ScanPosInside AND NOT "KukaRobot1_CtrlDB".sROBtoPLC.User.Cycle.DO241_SPalletPickInside AND NOT "KukaRobot1_CtrlDB".sROBtoPLC.User.Cycle.DO249_ShaftScanPutInside AND NOT "KukaRobot1_CtrlDB".sROBtoPLC.User.Cycle.DO253_SScanPickInside AND NOT "KukaRobot1_CtrlDB".sROBtoPLC.User.Cycle.DO257_TablePickInside AND NOT "KukaRobot1_CtrlDB".sROBtoPLC.User.Cycle.DO261_RingScanInside AND NOT "KukaRobot1_CtrlDB".sROBtoPLC.User.Cycle.DO265_LoadNGInside AND NOT "KukaRobot1_CtrlDB".sROBtoPLC.User.Cycle.DO273_PressShaftPutInside AND NOT "KukaRobot1_CtrlDB".sROBtoPLC.User.Cycle.DO277_PressRingPutInside AND NOT "KukaRobot1_CtrlDB".sROBtoPLC.User.Cycle.DO289_GluePutInside AND NOT "KukaRobot1_CtrlDB".sROBtoPLC.User.Cycle.DO305_GripScanInside AND NOT "KukaRobot1_CtrlDB".sROBtoPLC.User.Cycle.DO300_HomeInside;
END_REGION

REGION Network 18: Robot1 area
   RUNG wire#powerrail
      Contact( "AlwaysTRUE" )
      Contact( "KukaRobot1_CtrlDB".sROBtoPLC.User.Home.DO180_Robot2Area )
      Coil( "KukaRobot2_CtrlDB".sPLCtoROB.User.Home.DI170 )
   END_RUNG
   // the same network as SCL:
   "KukaRobot2_CtrlDB".sPLCtoROB.User.Home.DI170 := "AlwaysTRUE" AND "KukaRobot1_CtrlDB".sROBtoPLC.User.Home.DO180_Robot2Area;
END_REGION

REGION Network 19: MasteringTest_Req & BrakeTest_Req
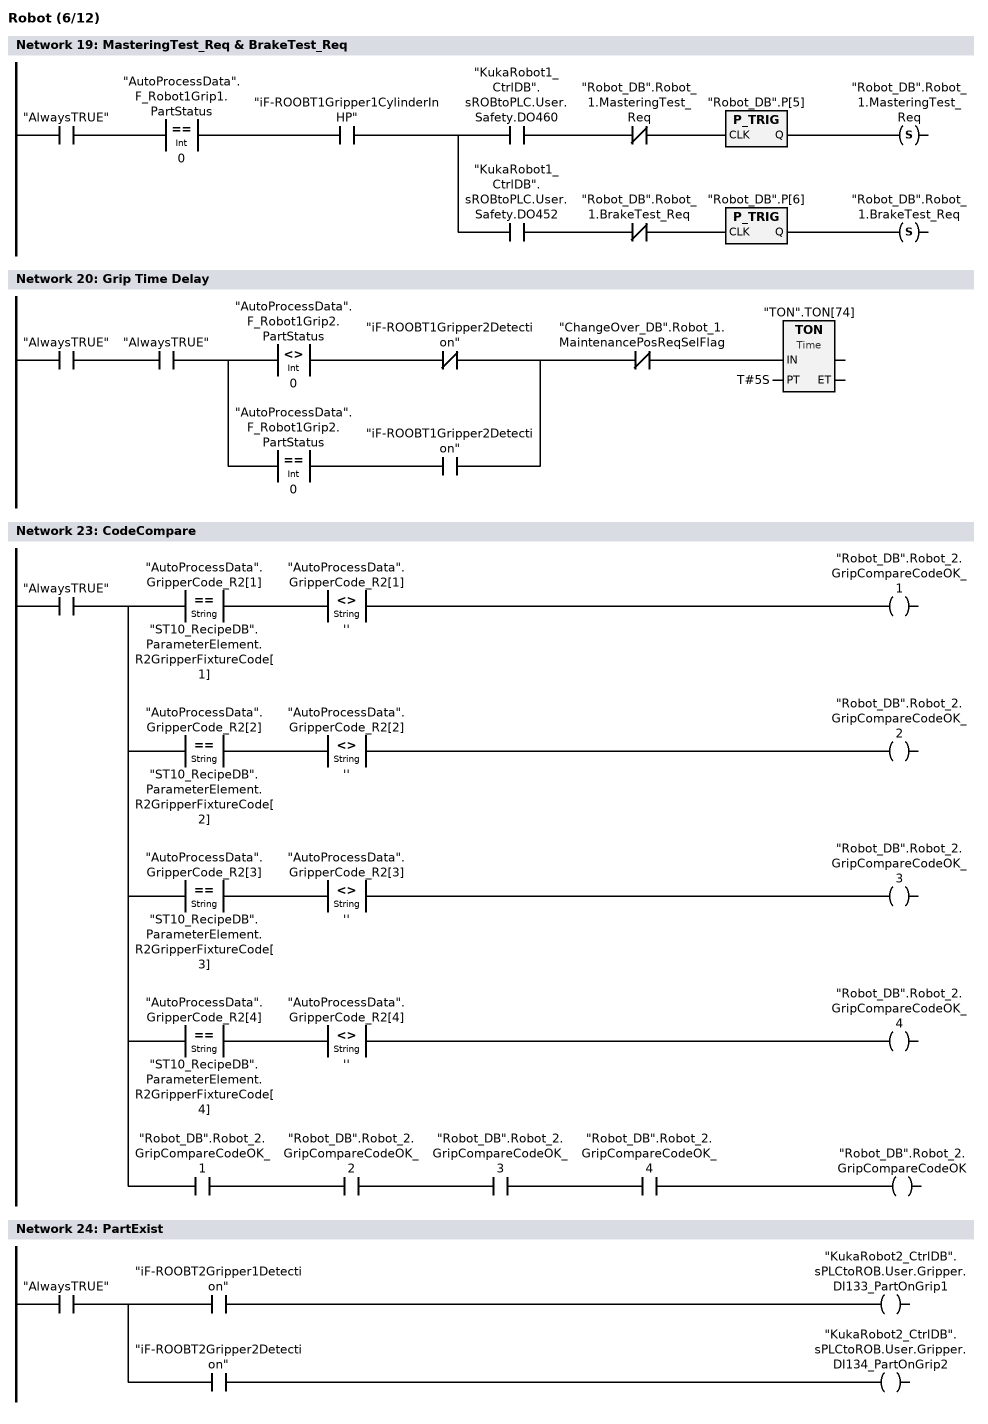
   RUNG wire#powerrail
      Contact( "AlwaysTRUE" )
      { S7_Templates := "SrcType := Int" } EQ_Contact(in1 := "AutoProcessData".F_Robot1Grip1.PartStatus, in2 := 0)
      Contact( "iF-ROOBT1Gripper1CylinderInHP" )
      wire#w1
      Contact( "KukaRobot1_CtrlDB".sROBtoPLC.User.Safety.DO460 )
      I_Contact( "Robot_DB".Robot_1.MasteringTest_Req )
      P_Trig( "Robot_DB".P[5] )
      S_Coil( "Robot_DB".Robot_1.MasteringTest_Req )
   END_RUNG
   RUNG wire#w1
      Contact( "KukaRobot1_CtrlDB".sROBtoPLC.User.Safety.DO452 )
      I_Contact( "Robot_DB".Robot_1.BrakeTest_Req )
      P_Trig( "Robot_DB".P[6] )
      S_Coil( "Robot_DB".Robot_1.BrakeTest_Req )
   END_RUNG
   // the same network as SCL:
   #_w1 := "AlwaysTRUE" AND ("AutoProcessData".F_Robot1Grip1.PartStatus = 0) AND "iF-ROOBT1Gripper1CylinderInHP";
   #_w2 := #_w1 AND "KukaRobot1_CtrlDB".sROBtoPLC.User.Safety.DO460 AND NOT "Robot_DB".Robot_1.MasteringTest_Req;
   #_w3 := #_w2 AND NOT "Robot_DB".P[5];   // rising edge
   "Robot_DB".P[5] := #_w2;
   IF #_w3 THEN "Robot_DB".Robot_1.MasteringTest_Req := TRUE; END_IF;
   #_w4 := #_w1 AND "KukaRobot1_CtrlDB".sROBtoPLC.User.Safety.DO452 AND NOT "Robot_DB".Robot_1.BrakeTest_Req;
   #_w5 := #_w4 AND NOT "Robot_DB".P[6];   // rising edge
   "Robot_DB".P[6] := #_w4;
   IF #_w5 THEN "Robot_DB".Robot_1.BrakeTest_Req := TRUE; END_IF;
END_REGION

REGION Network 20: Grip Time Delay
   RUNG wire#powerrail
      Contact( "AlwaysTRUE" )
      Contact( "AlwaysTRUE" )
      wire#w1
      { S7_Templates := "SrcType := Int" } NE_Contact(in1 := "AutoProcessData".F_Robot1Grip2.PartStatus, in2 := 0)
      I_Contact( "iF-ROOBT1Gripper2Detection" )
      wire#w2
      I_Contact( "ChangeOver_DB".Robot_1.MaintenancePosReqSelFlag )
      { S7_Templates := "time_type := Time" } "TON".TON[74].TON(pt := T#5S, et =>)
   END_RUNG
   RUNG wire#w1
      { S7_Templates := "SrcType := Int" } EQ_Contact(in1 := "AutoProcessData".F_Robot1Grip2.PartStatus, in2 := 0)
      Contact( "iF-ROOBT1Gripper2Detection" )
   END_RUNG wire#w2
   // the same network as SCL:
   "TON".TON[74].TON(IN := "AlwaysTRUE" AND "AlwaysTRUE" AND ((("AutoProcessData".F_Robot1Grip2.PartStatus <> 0) AND NOT "iF-ROOBT1Gripper2Detection") OR (("AutoProcessData".F_Robot1Grip2.PartStatus = 0) AND "iF-ROOBT1Gripper2Detection")) AND NOT "ChangeOver_DB".Robot_1.MaintenancePosReqSelFlag,
                     PT := T#5S);
END_REGION

REGION Network 22: ----------------------------------------- Robot_2 -------------------------------------
END_REGION

REGION Network 23: CodeCompare
   RUNG wire#powerrail
      Contact( "AlwaysTRUE" )
      wire#w1
      { S7_Templates := "SrcType := String" } EQ_Contact(in1 := "AutoProcessData".GripperCode_R2[1], in2 := "ST10_RecipeDB".ParameterElement.R2GripperFixtureCode[1])
      { S7_Templates := "SrcType := String" } NE_Contact(in1 := "AutoProcessData".GripperCode_R2[1], in2 := '')
      Coil( "Robot_DB".Robot_2.GripCompareCodeOK_1 )
   END_RUNG
   RUNG wire#w1
      { S7_Templates := "SrcType := String" } EQ_Contact(in1 := "AutoProcessData".GripperCode_R2[2], in2 := "ST10_RecipeDB".ParameterElement.R2GripperFixtureCode[2])
      { S7_Templates := "SrcType := String" } NE_Contact(in1 := "AutoProcessData".GripperCode_R2[2], in2 := '')
      Coil( "Robot_DB".Robot_2.GripCompareCodeOK_2 )
   END_RUNG
   RUNG wire#w1
      { S7_Templates := "SrcType := String" } EQ_Contact(in1 := "AutoProcessData".GripperCode_R2[3], in2 := "ST10_RecipeDB".ParameterElement.R2GripperFixtureCode[3])
      { S7_Templates := "SrcType := String" } NE_Contact(in1 := "AutoProcessData".GripperCode_R2[3], in2 := '')
      Coil( "Robot_DB".Robot_2.GripCompareCodeOK_3 )
   END_RUNG
   RUNG wire#w1
      { S7_Templates := "SrcType := String" } EQ_Contact(in1 := "AutoProcessData".GripperCode_R2[4], in2 := "ST10_RecipeDB".ParameterElement.R2GripperFixtureCode[4])
      { S7_Templates := "SrcType := String" } NE_Contact(in1 := "AutoProcessData".GripperCode_R2[4], in2 := '')
      Coil( "Robot_DB".Robot_2.GripCompareCodeOK_4 )
   END_RUNG
   RUNG wire#w1
      Contact( "Robot_DB".Robot_2.GripCompareCodeOK_1 )
      Contact( "Robot_DB".Robot_2.GripCompareCodeOK_2 )
      Contact( "Robot_DB".Robot_2.GripCompareCodeOK_3 )
      Contact( "Robot_DB".Robot_2.GripCompareCodeOK_4 )
      Coil( "Robot_DB".Robot_2.GripCompareCodeOK )
   END_RUNG
   // the same network as SCL:
   "Robot_DB".Robot_2.GripCompareCodeOK_1 := "AlwaysTRUE" AND ("AutoProcessData".GripperCode_R2[1] = "ST10_RecipeDB".ParameterElement.R2GripperFixtureCode[1]) AND ("AutoProcessData".GripperCode_R2[1] <> '');
   "Robot_DB".Robot_2.GripCompareCodeOK_2 := "AlwaysTRUE" AND ("AutoProcessData".GripperCode_R2[2] = "ST10_RecipeDB".ParameterElement.R2GripperFixtureCode[2]) AND ("AutoProcessData".GripperCode_R2[2] <> '');
   "Robot_DB".Robot_2.GripCompareCodeOK_3 := "AlwaysTRUE" AND ("AutoProcessData".GripperCode_R2[3] = "ST10_RecipeDB".ParameterElement.R2GripperFixtureCode[3]) AND ("AutoProcessData".GripperCode_R2[3] <> '');
   "Robot_DB".Robot_2.GripCompareCodeOK_4 := "AlwaysTRUE" AND ("AutoProcessData".GripperCode_R2[4] = "ST10_RecipeDB".ParameterElement.R2GripperFixtureCode[4]) AND ("AutoProcessData".GripperCode_R2[4] <> '');
   "Robot_DB".Robot_2.GripCompareCodeOK := "AlwaysTRUE" AND "Robot_DB".Robot_2.GripCompareCodeOK_1 AND "Robot_DB".Robot_2.GripCompareCodeOK_2 AND "Robot_DB".Robot_2.GripCompareCodeOK_3 AND "Robot_DB".Robot_2.GripCompareCodeOK_4;
END_REGION

REGION Network 24: PartExist
   RUNG wire#powerrail
      Contact( "AlwaysTRUE" )
      wire#w1
      Contact( "iF-ROOBT2Gripper1Detection" )
      Coil( "KukaRobot2_CtrlDB".sPLCtoROB.User.Gripper.DI133_PartOnGrip1 )
   END_RUNG
   RUNG wire#w1
      Contact( "iF-ROOBT2Gripper2Detection" )
      Coil( "KukaRobot2_CtrlDB".sPLCtoROB.User.Gripper.DI134_PartOnGrip2 )
   END_RUNG
   // the same network as SCL:
   "KukaRobot2_CtrlDB".sPLCtoROB.User.Gripper.DI133_PartOnGrip1 := "AlwaysTRUE" AND "iF-ROOBT2Gripper1Detection";
   "KukaRobot2_CtrlDB".sPLCtoROB.User.Gripper.DI134_PartOnGrip2 := "AlwaysTRUE" AND "iF-ROOBT2Gripper2Detection";
END_REGION

REGION Network 25: SpeedCount
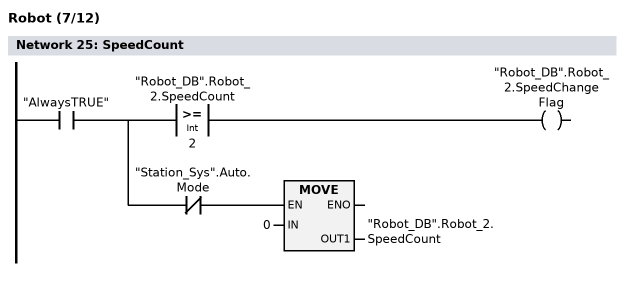
   RUNG wire#powerrail
      Contact( "AlwaysTRUE" )
      wire#w1
      { S7_Templates := "SrcType := Int" } GE_Contact(in1 := "Robot_DB".Robot_2.SpeedCount, in2 := 2)
      Coil( "Robot_DB".Robot_2.SpeedChangeFlag )
   END_RUNG
   RUNG wire#w1
      I_Contact( "Station_Sys".Auto.Mode )
      Move(in := 0, out1 => "Robot_DB".Robot_2.SpeedCount)
   END_RUNG
   // the same network as SCL:
   "Robot_DB".Robot_2.SpeedChangeFlag := "AlwaysTRUE" AND ("Robot_DB".Robot_2.SpeedCount >= 2);
   IF "AlwaysTRUE" AND NOT "Station_Sys".Auto.Mode THEN "Robot_DB".Robot_2.SpeedCount := 0; END_IF;
END_REGION

REGION Network 26: Robot2Speed Interlock
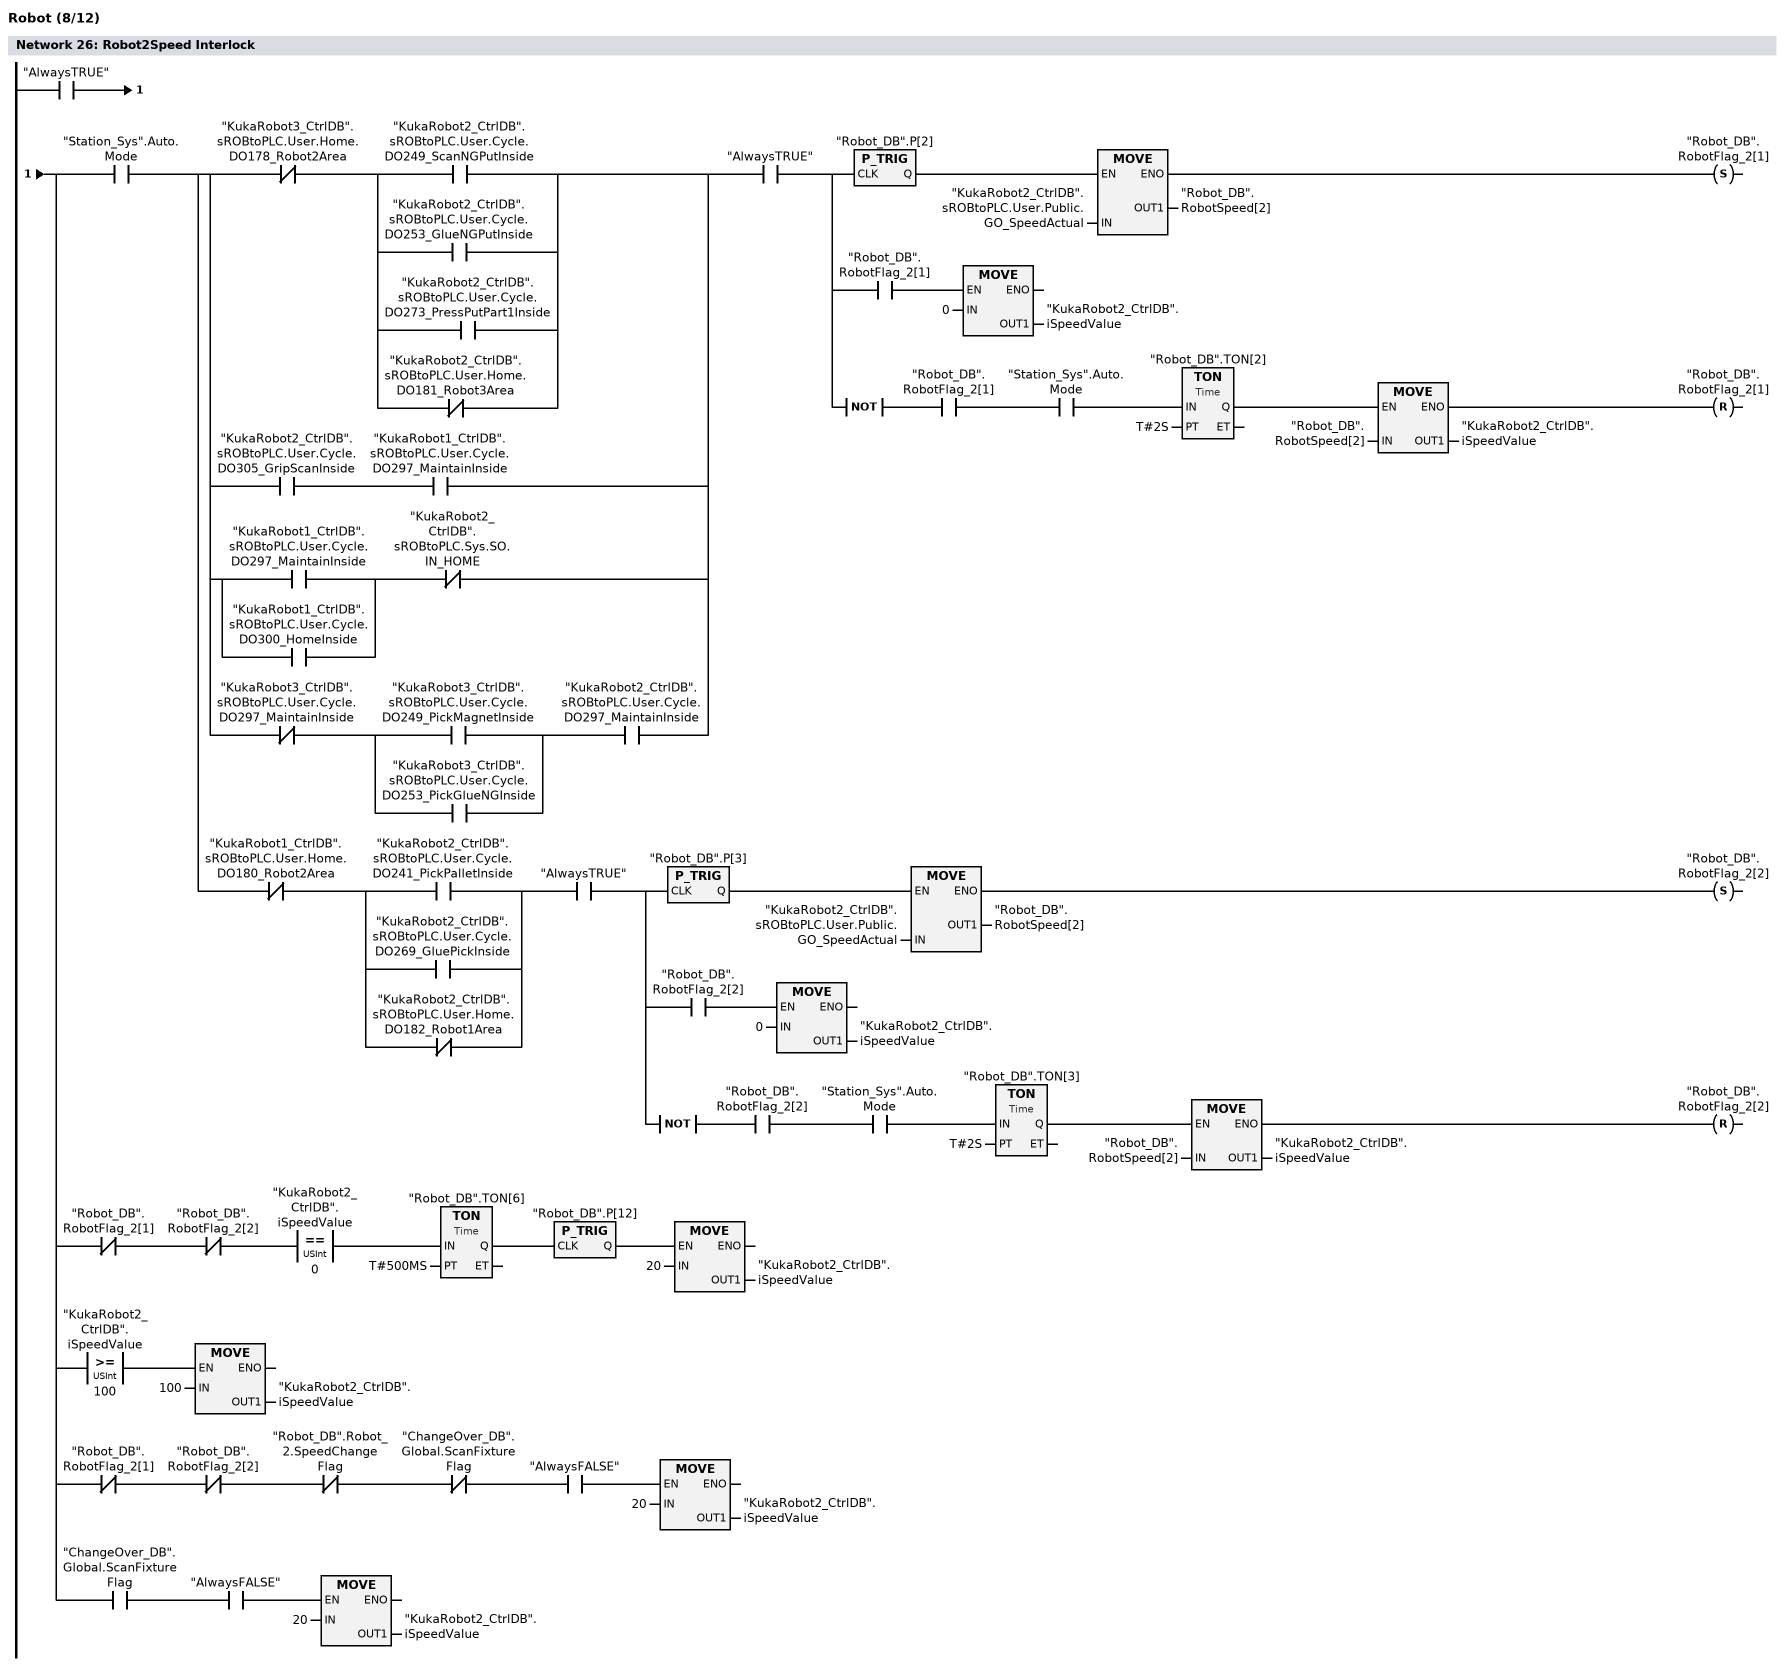
   RUNG wire#powerrail
      Contact( "AlwaysTRUE" )
      wire#w1
      Contact( "Station_Sys".Auto.Mode )
      wire#w2
      I_Contact( "KukaRobot3_CtrlDB".sROBtoPLC.User.Home.DO178_Robot2Area )
      wire#w3
      Contact( "KukaRobot2_CtrlDB".sROBtoPLC.User.Cycle.DO249_ScanNGPutInside )
      wire#w4
      Contact( "AlwaysTRUE" )
      wire#w8
      P_Trig( "Robot_DB".P[2] )
      Move(in := "KukaRobot2_CtrlDB".sROBtoPLC.User.Public.GO_SpeedActual, out1 => "Robot_DB".RobotSpeed[2])
      S_Coil( "Robot_DB".RobotFlag_2[1] )
   END_RUNG
   RUNG wire#w3
      Contact( "KukaRobot2_CtrlDB".sROBtoPLC.User.Cycle.DO253_GlueNGPutInside )
   END_RUNG wire#w4
   RUNG wire#w3
      Contact( "KukaRobot2_CtrlDB".sROBtoPLC.User.Cycle.DO273_PressPutPart1Inside )
   END_RUNG wire#w4
   RUNG wire#w3
      I_Contact( "KukaRobot2_CtrlDB".sROBtoPLC.User.Home.DO181_Robot3Area )
   END_RUNG wire#w4
   RUNG wire#w2
      Contact( "KukaRobot2_CtrlDB".sROBtoPLC.User.Cycle.DO305_GripScanInside )
      Contact( "KukaRobot1_CtrlDB".sROBtoPLC.User.Cycle.DO297_MaintainInside )
   END_RUNG wire#w4
   RUNG wire#w2
      Contact( "KukaRobot1_CtrlDB".sROBtoPLC.User.Cycle.DO297_MaintainInside )
      wire#w5
      I_Contact( "KukaRobot2_CtrlDB".sROBtoPLC.Sys.SO.IN_HOME )
   END_RUNG wire#w4
   RUNG wire#w2
      Contact( "KukaRobot1_CtrlDB".sROBtoPLC.User.Cycle.DO300_HomeInside )
   END_RUNG wire#w5
   RUNG wire#w2
      I_Contact( "KukaRobot3_CtrlDB".sROBtoPLC.User.Cycle.DO297_MaintainInside )
      wire#w6
      Contact( "KukaRobot3_CtrlDB".sROBtoPLC.User.Cycle.DO249_PickMagnetInside )
      wire#w7
      Contact( "KukaRobot2_CtrlDB".sROBtoPLC.User.Cycle.DO297_MaintainInside )
   END_RUNG wire#w4
   RUNG wire#w6
      Contact( "KukaRobot3_CtrlDB".sROBtoPLC.User.Cycle.DO253_PickGlueNGInside )
   END_RUNG wire#w7
   RUNG wire#w8
      Contact( "Robot_DB".RobotFlag_2[1] )
      Move(in := 0, out1 => "KukaRobot2_CtrlDB".iSpeedValue)
   END_RUNG
   RUNG wire#w8
      Not()
      Contact( "Robot_DB".RobotFlag_2[1] )
      Contact( "Station_Sys".Auto.Mode )
      { S7_Templates := "time_type := Time" } "Robot_DB".TON[2].TON(pt := T#2S, et =>)
      Move(in := "Robot_DB".RobotSpeed[2], out1 => "KukaRobot2_CtrlDB".iSpeedValue)
      R_Coil( "Robot_DB".RobotFlag_2[1] )
   END_RUNG
   RUNG wire#w2
      I_Contact( "KukaRobot1_CtrlDB".sROBtoPLC.User.Home.DO180_Robot2Area )
      wire#w9
      Contact( "KukaRobot2_CtrlDB".sROBtoPLC.User.Cycle.DO241_PickPalletInside )
      wire#w10
      Contact( "AlwaysTRUE" )
      wire#w11
      P_Trig( "Robot_DB".P[3] )
      Move(in := "KukaRobot2_CtrlDB".sROBtoPLC.User.Public.GO_SpeedActual, out1 => "Robot_DB".RobotSpeed[2])
      S_Coil( "Robot_DB".RobotFlag_2[2] )
   END_RUNG
   RUNG wire#w9
      Contact( "KukaRobot2_CtrlDB".sROBtoPLC.User.Cycle.DO269_GluePickInside )
   END_RUNG wire#w10
   RUNG wire#w9
      I_Contact( "KukaRobot2_CtrlDB".sROBtoPLC.User.Home.DO182_Robot1Area )
   END_RUNG wire#w10
   RUNG wire#w11
      Contact( "Robot_DB".RobotFlag_2[2] )
      Move(in := 0, out1 => "KukaRobot2_CtrlDB".iSpeedValue)
   END_RUNG
   RUNG wire#w11
      Not()
      Contact( "Robot_DB".RobotFlag_2[2] )
      Contact( "Station_Sys".Auto.Mode )
      { S7_Templates := "time_type := Time" } "Robot_DB".TON[3].TON(pt := T#2S, et =>)
      Move(in := "Robot_DB".RobotSpeed[2], out1 => "KukaRobot2_CtrlDB".iSpeedValue)
      R_Coil( "Robot_DB".RobotFlag_2[2] )
   END_RUNG
   RUNG wire#w1
      I_Contact( "Robot_DB".RobotFlag_2[1] )
      I_Contact( "Robot_DB".RobotFlag_2[2] )
      { S7_Templates := "SrcType := USInt" } EQ_Contact(in1 := "KukaRobot2_CtrlDB".iSpeedValue, in2 := 0)
      { S7_Templates := "time_type := Time" } "Robot_DB".TON[6].TON(pt := T#500MS, et =>)
      P_Trig( "Robot_DB".P[12] )
      Move(in := 20, out1 => "KukaRobot2_CtrlDB".iSpeedValue)
   END_RUNG
   RUNG wire#w1
      { S7_Templates := "SrcType := USInt" } GE_Contact(in1 := "KukaRobot2_CtrlDB".iSpeedValue, in2 := 100)
      Move(in := 100, out1 => "KukaRobot2_CtrlDB".iSpeedValue)
   END_RUNG
   RUNG wire#w1
      I_Contact( "Robot_DB".RobotFlag_2[1] )
      I_Contact( "Robot_DB".RobotFlag_2[2] )
      I_Contact( "Robot_DB".Robot_2.SpeedChangeFlag )
      I_Contact( "ChangeOver_DB".Global.ScanFixtureFlag )
      Contact( "AlwaysFALSE" )
      Move(in := 20, out1 => "KukaRobot2_CtrlDB".iSpeedValue)
   END_RUNG
   RUNG wire#w1
      Contact( "ChangeOver_DB".Global.ScanFixtureFlag )
      Contact( "AlwaysFALSE" )
      Move(in := 20, out1 => "KukaRobot2_CtrlDB".iSpeedValue)
   END_RUNG
   // the same network as SCL:
   #_w1 := "AlwaysTRUE" AND "Station_Sys".Auto.Mode;
   #_w2 := #_w1 AND ((NOT "KukaRobot3_CtrlDB".sROBtoPLC.User.Home.DO178_Robot2Area AND ("KukaRobot2_CtrlDB".sROBtoPLC.User.Cycle.DO249_ScanNGPutInside OR "KukaRobot2_CtrlDB".sROBtoPLC.User.Cycle.DO253_GlueNGPutInside OR "KukaRobot2_CtrlDB".sROBtoPLC.User.Cycle.DO273_PressPutPart1Inside OR NOT "KukaRobot2_CtrlDB".sROBtoPLC.User.Home.DO181_Robot3Area)) OR ("KukaRobot2_CtrlDB".sROBtoPLC.User.Cycle.DO305_GripScanInside AND "KukaRobot1_CtrlDB".sROBtoPLC.User.Cycle.DO297_MaintainInside) OR (("KukaRobot1_CtrlDB".sROBtoPLC.User.Cycle.DO297_MaintainInside OR "KukaRobot1_CtrlDB".sROBtoPLC.User.Cycle.DO300_HomeInside) AND NOT "KukaRobot2_CtrlDB".sROBtoPLC.Sys.SO.IN_HOME) OR (NOT "KukaRobot3_CtrlDB".sROBtoPLC.User.Cycle.DO297_MaintainInside AND ("KukaRobot3_CtrlDB".sROBtoPLC.User.Cycle.DO249_PickMagnetInside OR "KukaRobot3_CtrlDB".sROBtoPLC.User.Cycle.DO253_PickGlueNGInside) AND "KukaRobot2_CtrlDB".sROBtoPLC.User.Cycle.DO297_MaintainInside)) AND "AlwaysTRUE";
   #_w3 := #_w2 AND NOT "Robot_DB".P[2];   // rising edge
   "Robot_DB".P[2] := #_w2;
   IF #_w3 THEN
       "Robot_DB".RobotSpeed[2] := "KukaRobot2_CtrlDB".sROBtoPLC.User.Public.GO_SpeedActual;
       "Robot_DB".RobotFlag_2[1] := TRUE;
   END_IF;
   IF #_w2 AND "Robot_DB".RobotFlag_2[1] THEN "KukaRobot2_CtrlDB".iSpeedValue := 0; END_IF;
   "Robot_DB".TON[2].TON(IN := NOT #_w2 AND "Robot_DB".RobotFlag_2[1] AND "Station_Sys".Auto.Mode, PT := T#2S);
   IF "Robot_DB".TON[2].Q THEN
       "KukaRobot2_CtrlDB".iSpeedValue := "Robot_DB".RobotSpeed[2];
       "Robot_DB".RobotFlag_2[1] := FALSE;
   END_IF;
   #_w4 := #_w1 AND NOT "KukaRobot1_CtrlDB".sROBtoPLC.User.Home.DO180_Robot2Area AND ("KukaRobot2_CtrlDB".sROBtoPLC.User.Cycle.DO241_PickPalletInside OR "KukaRobot2_CtrlDB".sROBtoPLC.User.Cycle.DO269_GluePickInside OR NOT "KukaRobot2_CtrlDB".sROBtoPLC.User.Home.DO182_Robot1Area) AND "AlwaysTRUE";
   #_w5 := #_w4 AND NOT "Robot_DB".P[3];   // rising edge
   "Robot_DB".P[3] := #_w4;
   IF #_w5 THEN
       "Robot_DB".RobotSpeed[2] := "KukaRobot2_CtrlDB".sROBtoPLC.User.Public.GO_SpeedActual;
       "Robot_DB".RobotFlag_2[2] := TRUE;
   END_IF;
   IF #_w4 AND "Robot_DB".RobotFlag_2[2] THEN "KukaRobot2_CtrlDB".iSpeedValue := 0; END_IF;
   "Robot_DB".TON[3].TON(IN := NOT #_w4 AND "Robot_DB".RobotFlag_2[2] AND "Station_Sys".Auto.Mode, PT := T#2S);
   IF "Robot_DB".TON[3].Q THEN
       "KukaRobot2_CtrlDB".iSpeedValue := "Robot_DB".RobotSpeed[2];
       "Robot_DB".RobotFlag_2[2] := FALSE;
   END_IF;
   "Robot_DB".TON[6].TON(IN := "AlwaysTRUE" AND NOT "Robot_DB".RobotFlag_2[1] AND NOT "Robot_DB".RobotFlag_2[2] AND ("KukaRobot2_CtrlDB".iSpeedValue = 0),
                         PT := T#500MS);
   #_w6 := "Robot_DB".TON[6].Q AND NOT "Robot_DB".P[12];   // rising edge
   "Robot_DB".P[12] := "Robot_DB".TON[6].Q;
   IF #_w6 THEN "KukaRobot2_CtrlDB".iSpeedValue := 20; END_IF;
   IF "AlwaysTRUE" AND ("KukaRobot2_CtrlDB".iSpeedValue >= 100) THEN
       "KukaRobot2_CtrlDB".iSpeedValue := 100;
   END_IF;
   IF "AlwaysTRUE" AND NOT "Robot_DB".RobotFlag_2[1] AND NOT "Robot_DB".RobotFlag_2[2] AND NOT "Robot_DB".Robot_2.SpeedChangeFlag AND NOT "ChangeOver_DB".Global.ScanFixtureFlag AND "AlwaysFALSE" THEN
       "KukaRobot2_CtrlDB".iSpeedValue := 20;
   END_IF;
   IF "AlwaysTRUE" AND "ChangeOver_DB".Global.ScanFixtureFlag AND "AlwaysFALSE" THEN
       "KukaRobot2_CtrlDB".iSpeedValue := 20;
   END_IF;
END_REGION

REGION Network 27: Robot2 No Task Running
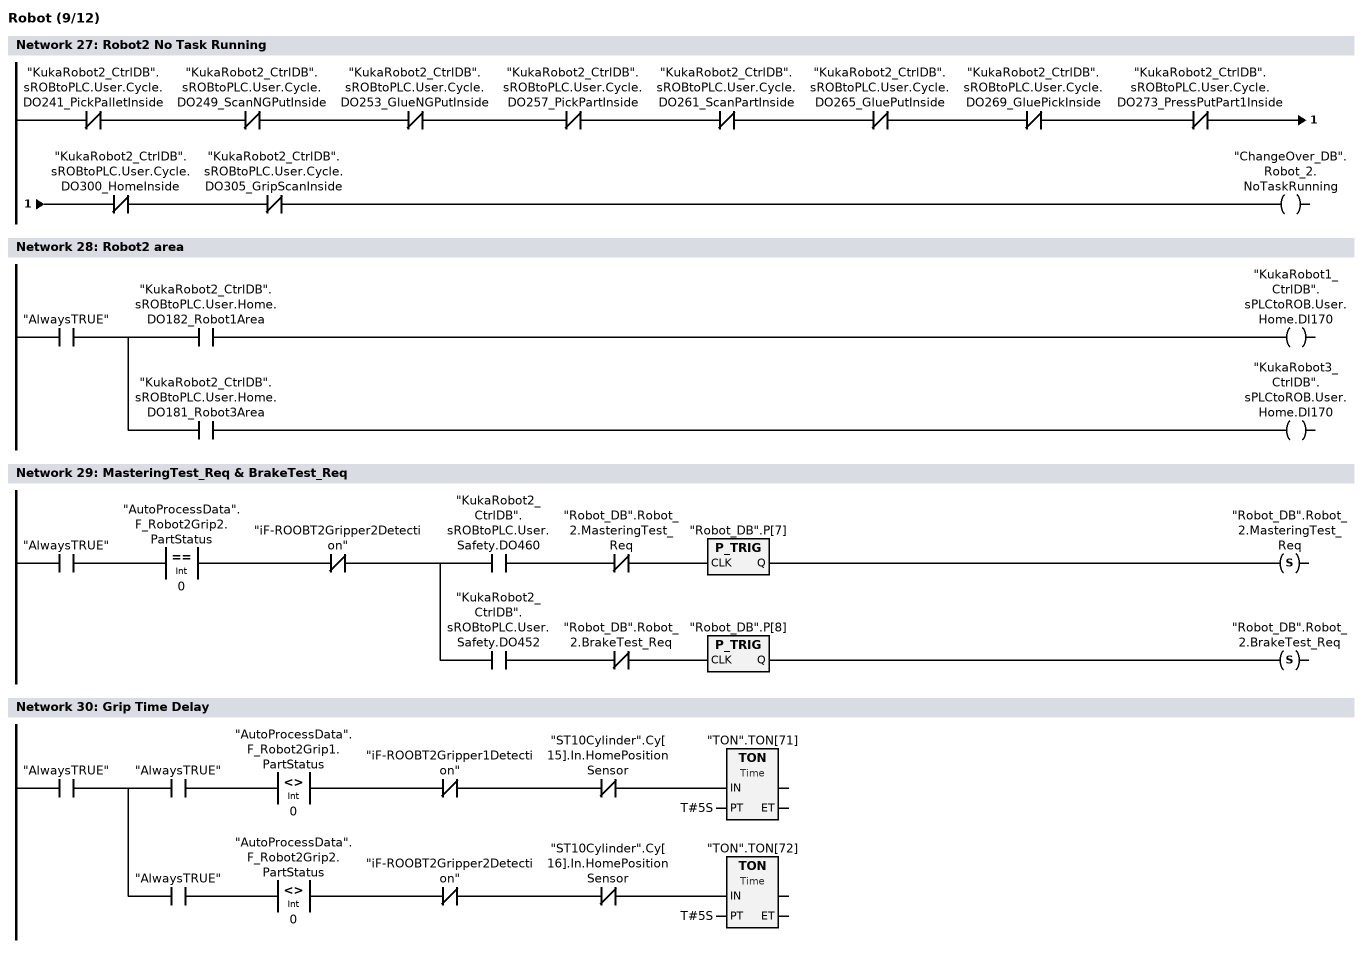
   RUNG wire#powerrail
      I_Contact( "KukaRobot2_CtrlDB".sROBtoPLC.User.Cycle.DO241_PickPalletInside )
      I_Contact( "KukaRobot2_CtrlDB".sROBtoPLC.User.Cycle.DO249_ScanNGPutInside )
      I_Contact( "KukaRobot2_CtrlDB".sROBtoPLC.User.Cycle.DO253_GlueNGPutInside )
      I_Contact( "KukaRobot2_CtrlDB".sROBtoPLC.User.Cycle.DO257_PickPartInside )
      I_Contact( "KukaRobot2_CtrlDB".sROBtoPLC.User.Cycle.DO261_ScanPartInside )
      I_Contact( "KukaRobot2_CtrlDB".sROBtoPLC.User.Cycle.DO265_GluePutInside )
      I_Contact( "KukaRobot2_CtrlDB".sROBtoPLC.User.Cycle.DO269_GluePickInside )
      I_Contact( "KukaRobot2_CtrlDB".sROBtoPLC.User.Cycle.DO273_PressPutPart1Inside )
      I_Contact( "KukaRobot2_CtrlDB".sROBtoPLC.User.Cycle.DO300_HomeInside )
      I_Contact( "KukaRobot2_CtrlDB".sROBtoPLC.User.Cycle.DO305_GripScanInside )
      Coil( "ChangeOver_DB".Robot_2.NoTaskRunning )
   END_RUNG
   // the same network as SCL:
   "ChangeOver_DB".Robot_2.NoTaskRunning := NOT "KukaRobot2_CtrlDB".sROBtoPLC.User.Cycle.DO241_PickPalletInside AND NOT "KukaRobot2_CtrlDB".sROBtoPLC.User.Cycle.DO249_ScanNGPutInside AND NOT "KukaRobot2_CtrlDB".sROBtoPLC.User.Cycle.DO253_GlueNGPutInside AND NOT "KukaRobot2_CtrlDB".sROBtoPLC.User.Cycle.DO257_PickPartInside AND NOT "KukaRobot2_CtrlDB".sROBtoPLC.User.Cycle.DO261_ScanPartInside AND NOT "KukaRobot2_CtrlDB".sROBtoPLC.User.Cycle.DO265_GluePutInside AND NOT "KukaRobot2_CtrlDB".sROBtoPLC.User.Cycle.DO269_GluePickInside AND NOT "KukaRobot2_CtrlDB".sROBtoPLC.User.Cycle.DO273_PressPutPart1Inside AND NOT "KukaRobot2_CtrlDB".sROBtoPLC.User.Cycle.DO300_HomeInside AND NOT "KukaRobot2_CtrlDB".sROBtoPLC.User.Cycle.DO305_GripScanInside;
END_REGION

REGION Network 28: Robot2 area
   RUNG wire#powerrail
      Contact( "AlwaysTRUE" )
      wire#w1
      Contact( "KukaRobot2_CtrlDB".sROBtoPLC.User.Home.DO182_Robot1Area )
      Coil( "KukaRobot1_CtrlDB".sPLCtoROB.User.Home.DI170 )
   END_RUNG
   RUNG wire#w1
      Contact( "KukaRobot2_CtrlDB".sROBtoPLC.User.Home.DO181_Robot3Area )
      Coil( "KukaRobot3_CtrlDB".sPLCtoROB.User.Home.DI170 )
   END_RUNG
   // the same network as SCL:
   "KukaRobot1_CtrlDB".sPLCtoROB.User.Home.DI170 := "AlwaysTRUE" AND "KukaRobot2_CtrlDB".sROBtoPLC.User.Home.DO182_Robot1Area;
   "KukaRobot3_CtrlDB".sPLCtoROB.User.Home.DI170 := "AlwaysTRUE" AND "KukaRobot2_CtrlDB".sROBtoPLC.User.Home.DO181_Robot3Area;
END_REGION

REGION Network 29: MasteringTest_Req & BrakeTest_Req
   RUNG wire#powerrail
      Contact( "AlwaysTRUE" )
      { S7_Templates := "SrcType := Int" } EQ_Contact(in1 := "AutoProcessData".F_Robot2Grip2.PartStatus, in2 := 0)
      I_Contact( "iF-ROOBT2Gripper2Detection" )
      wire#w1
      Contact( "KukaRobot2_CtrlDB".sROBtoPLC.User.Safety.DO460 )
      I_Contact( "Robot_DB".Robot_2.MasteringTest_Req )
      P_Trig( "Robot_DB".P[7] )
      S_Coil( "Robot_DB".Robot_2.MasteringTest_Req )
   END_RUNG
   RUNG wire#w1
      Contact( "KukaRobot2_CtrlDB".sROBtoPLC.User.Safety.DO452 )
      I_Contact( "Robot_DB".Robot_2.BrakeTest_Req )
      P_Trig( "Robot_DB".P[8] )
      S_Coil( "Robot_DB".Robot_2.BrakeTest_Req )
   END_RUNG
   // the same network as SCL:
   #_w1 := "AlwaysTRUE" AND ("AutoProcessData".F_Robot2Grip2.PartStatus = 0) AND NOT "iF-ROOBT2Gripper2Detection";
   #_w2 := #_w1 AND "KukaRobot2_CtrlDB".sROBtoPLC.User.Safety.DO460 AND NOT "Robot_DB".Robot_2.MasteringTest_Req;
   #_w3 := #_w2 AND NOT "Robot_DB".P[7];   // rising edge
   "Robot_DB".P[7] := #_w2;
   IF #_w3 THEN "Robot_DB".Robot_2.MasteringTest_Req := TRUE; END_IF;
   #_w4 := #_w1 AND "KukaRobot2_CtrlDB".sROBtoPLC.User.Safety.DO452 AND NOT "Robot_DB".Robot_2.BrakeTest_Req;
   #_w5 := #_w4 AND NOT "Robot_DB".P[8];   // rising edge
   "Robot_DB".P[8] := #_w4;
   IF #_w5 THEN "Robot_DB".Robot_2.BrakeTest_Req := TRUE; END_IF;
END_REGION

REGION Network 30: Grip Time Delay
   RUNG wire#powerrail
      Contact( "AlwaysTRUE" )
      wire#w1
      Contact( "AlwaysTRUE" )
      { S7_Templates := "SrcType := Int" } NE_Contact(in1 := "AutoProcessData".F_Robot2Grip1.PartStatus, in2 := 0)
      I_Contact( "iF-ROOBT2Gripper1Detection" )
      I_Contact( "ST10Cylinder".Cy[15].In.HomePositionSensor )
      { S7_Templates := "time_type := Time" } "TON".TON[71].TON(pt := T#5S, et =>)
   END_RUNG
   RUNG wire#w1
      Contact( "AlwaysTRUE" )
      { S7_Templates := "SrcType := Int" } NE_Contact(in1 := "AutoProcessData".F_Robot2Grip2.PartStatus, in2 := 0)
      I_Contact( "iF-ROOBT2Gripper2Detection" )
      I_Contact( "ST10Cylinder".Cy[16].In.HomePositionSensor )
      { S7_Templates := "time_type := Time" } "TON".TON[72].TON(pt := T#5S, et =>)
   END_RUNG
   // the same network as SCL:
   "TON".TON[71].TON(IN := "AlwaysTRUE" AND "AlwaysTRUE" AND ("AutoProcessData".F_Robot2Grip1.PartStatus <> 0) AND NOT "iF-ROOBT2Gripper1Detection" AND NOT "ST10Cylinder".Cy[15].In.HomePositionSensor,
                     PT := T#5S);
   "TON".TON[72].TON(IN := "AlwaysTRUE" AND "AlwaysTRUE" AND ("AutoProcessData".F_Robot2Grip2.PartStatus <> 0) AND NOT "iF-ROOBT2Gripper2Detection" AND NOT "ST10Cylinder".Cy[16].In.HomePositionSensor,
                     PT := T#5S);
END_REGION

REGION Network 32: ----------------------------------------- Robot_3 -------------------------------------
END_REGION

REGION Network 33: CodeCompare
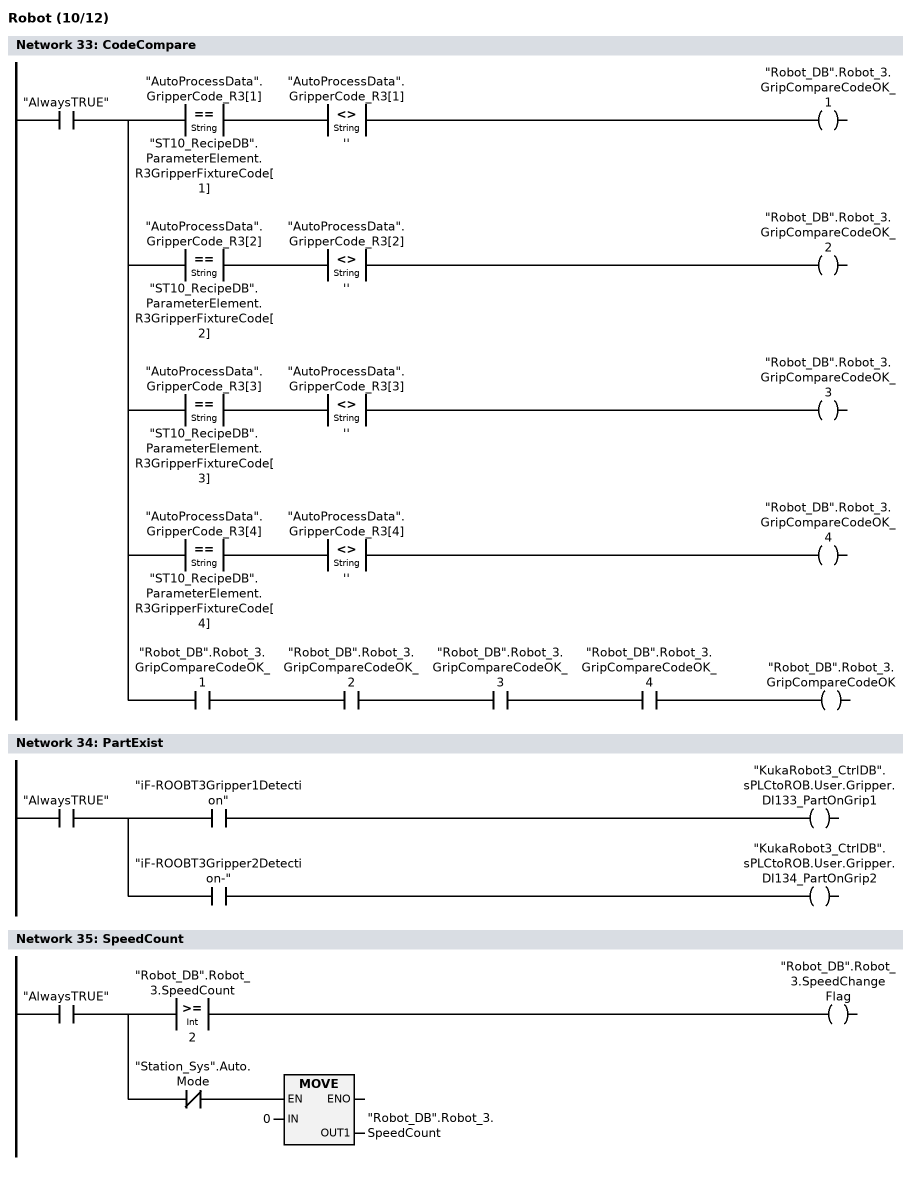
   RUNG wire#powerrail
      Contact( "AlwaysTRUE" )
      wire#w1
      { S7_Templates := "SrcType := String" } EQ_Contact(in1 := "AutoProcessData".GripperCode_R3[1], in2 := "ST10_RecipeDB".ParameterElement.R3GripperFixtureCode[1])
      { S7_Templates := "SrcType := String" } NE_Contact(in1 := "AutoProcessData".GripperCode_R3[1], in2 := '')
      Coil( "Robot_DB".Robot_3.GripCompareCodeOK_1 )
   END_RUNG
   RUNG wire#w1
      { S7_Templates := "SrcType := String" } EQ_Contact(in1 := "AutoProcessData".GripperCode_R3[2], in2 := "ST10_RecipeDB".ParameterElement.R3GripperFixtureCode[2])
      { S7_Templates := "SrcType := String" } NE_Contact(in1 := "AutoProcessData".GripperCode_R3[2], in2 := '')
      Coil( "Robot_DB".Robot_3.GripCompareCodeOK_2 )
   END_RUNG
   RUNG wire#w1
      { S7_Templates := "SrcType := String" } EQ_Contact(in1 := "AutoProcessData".GripperCode_R3[3], in2 := "ST10_RecipeDB".ParameterElement.R3GripperFixtureCode[3])
      { S7_Templates := "SrcType := String" } NE_Contact(in1 := "AutoProcessData".GripperCode_R3[3], in2 := '')
      Coil( "Robot_DB".Robot_3.GripCompareCodeOK_3 )
   END_RUNG
   RUNG wire#w1
      { S7_Templates := "SrcType := String" } EQ_Contact(in1 := "AutoProcessData".GripperCode_R3[4], in2 := "ST10_RecipeDB".ParameterElement.R3GripperFixtureCode[4])
      { S7_Templates := "SrcType := String" } NE_Contact(in1 := "AutoProcessData".GripperCode_R3[4], in2 := '')
      Coil( "Robot_DB".Robot_3.GripCompareCodeOK_4 )
   END_RUNG
   RUNG wire#w1
      Contact( "Robot_DB".Robot_3.GripCompareCodeOK_1 )
      Contact( "Robot_DB".Robot_3.GripCompareCodeOK_2 )
      Contact( "Robot_DB".Robot_3.GripCompareCodeOK_3 )
      Contact( "Robot_DB".Robot_3.GripCompareCodeOK_4 )
      Coil( "Robot_DB".Robot_3.GripCompareCodeOK )
   END_RUNG
   // the same network as SCL:
   "Robot_DB".Robot_3.GripCompareCodeOK_1 := "AlwaysTRUE" AND ("AutoProcessData".GripperCode_R3[1] = "ST10_RecipeDB".ParameterElement.R3GripperFixtureCode[1]) AND ("AutoProcessData".GripperCode_R3[1] <> '');
   "Robot_DB".Robot_3.GripCompareCodeOK_2 := "AlwaysTRUE" AND ("AutoProcessData".GripperCode_R3[2] = "ST10_RecipeDB".ParameterElement.R3GripperFixtureCode[2]) AND ("AutoProcessData".GripperCode_R3[2] <> '');
   "Robot_DB".Robot_3.GripCompareCodeOK_3 := "AlwaysTRUE" AND ("AutoProcessData".GripperCode_R3[3] = "ST10_RecipeDB".ParameterElement.R3GripperFixtureCode[3]) AND ("AutoProcessData".GripperCode_R3[3] <> '');
   "Robot_DB".Robot_3.GripCompareCodeOK_4 := "AlwaysTRUE" AND ("AutoProcessData".GripperCode_R3[4] = "ST10_RecipeDB".ParameterElement.R3GripperFixtureCode[4]) AND ("AutoProcessData".GripperCode_R3[4] <> '');
   "Robot_DB".Robot_3.GripCompareCodeOK := "AlwaysTRUE" AND "Robot_DB".Robot_3.GripCompareCodeOK_1 AND "Robot_DB".Robot_3.GripCompareCodeOK_2 AND "Robot_DB".Robot_3.GripCompareCodeOK_3 AND "Robot_DB".Robot_3.GripCompareCodeOK_4;
END_REGION

REGION Network 34: PartExist
   RUNG wire#powerrail
      Contact( "AlwaysTRUE" )
      wire#w1
      Contact( "iF-ROOBT3Gripper1Detection" )
      Coil( "KukaRobot3_CtrlDB".sPLCtoROB.User.Gripper.DI133_PartOnGrip1 )
   END_RUNG
   RUNG wire#w1
      Contact( "iF-ROOBT3Gripper2Detection-" )
      Coil( "KukaRobot3_CtrlDB".sPLCtoROB.User.Gripper.DI134_PartOnGrip2 )
   END_RUNG
   // the same network as SCL:
   "KukaRobot3_CtrlDB".sPLCtoROB.User.Gripper.DI133_PartOnGrip1 := "AlwaysTRUE" AND "iF-ROOBT3Gripper1Detection";
   "KukaRobot3_CtrlDB".sPLCtoROB.User.Gripper.DI134_PartOnGrip2 := "AlwaysTRUE" AND "iF-ROOBT3Gripper2Detection-";
END_REGION

REGION Network 35: SpeedCount
   RUNG wire#powerrail
      Contact( "AlwaysTRUE" )
      wire#w1
      { S7_Templates := "SrcType := Int" } GE_Contact(in1 := "Robot_DB".Robot_3.SpeedCount, in2 := 2)
      Coil( "Robot_DB".Robot_3.SpeedChangeFlag )
   END_RUNG
   RUNG wire#w1
      I_Contact( "Station_Sys".Auto.Mode )
      Move(in := 0, out1 => "Robot_DB".Robot_3.SpeedCount)
   END_RUNG
   // the same network as SCL:
   "Robot_DB".Robot_3.SpeedChangeFlag := "AlwaysTRUE" AND ("Robot_DB".Robot_3.SpeedCount >= 2);
   IF "AlwaysTRUE" AND NOT "Station_Sys".Auto.Mode THEN "Robot_DB".Robot_3.SpeedCount := 0; END_IF;
END_REGION

REGION Network 36: Robot3Speed Interlock
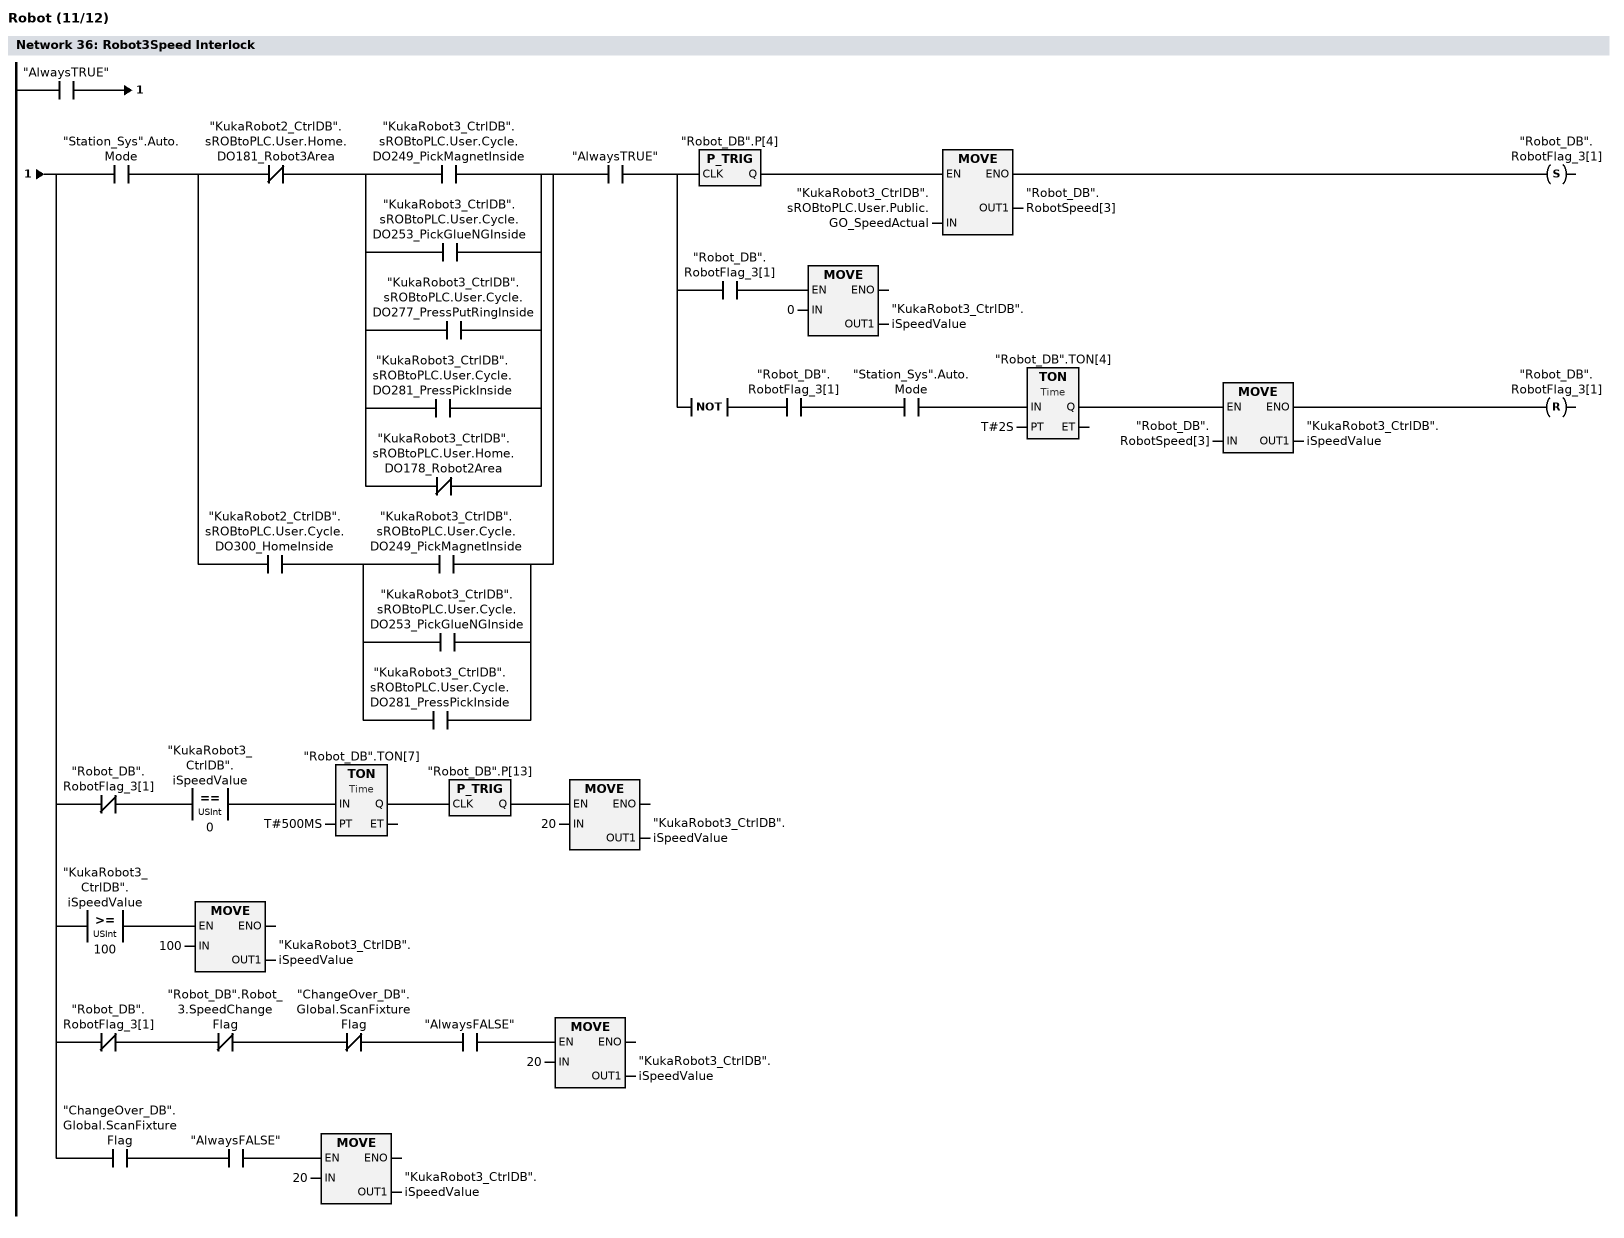
   RUNG wire#powerrail
      Contact( "AlwaysTRUE" )
      wire#w1
      Contact( "Station_Sys".Auto.Mode )
      wire#w2
      I_Contact( "KukaRobot2_CtrlDB".sROBtoPLC.User.Home.DO181_Robot3Area )
      wire#w3
      Contact( "KukaRobot3_CtrlDB".sROBtoPLC.User.Cycle.DO249_PickMagnetInside )
      wire#w4
      Contact( "AlwaysTRUE" )
      wire#w6
      P_Trig( "Robot_DB".P[4] )
      Move(in := "KukaRobot3_CtrlDB".sROBtoPLC.User.Public.GO_SpeedActual, out1 => "Robot_DB".RobotSpeed[3])
      S_Coil( "Robot_DB".RobotFlag_3[1] )
   END_RUNG
   RUNG wire#w3
      Contact( "KukaRobot3_CtrlDB".sROBtoPLC.User.Cycle.DO253_PickGlueNGInside )
   END_RUNG wire#w4
   RUNG wire#w3
      Contact( "KukaRobot3_CtrlDB".sROBtoPLC.User.Cycle.DO277_PressPutRingInside )
   END_RUNG wire#w4
   RUNG wire#w3
      Contact( "KukaRobot3_CtrlDB".sROBtoPLC.User.Cycle.DO281_PressPickInside )
   END_RUNG wire#w4
   RUNG wire#w3
      I_Contact( "KukaRobot3_CtrlDB".sROBtoPLC.User.Home.DO178_Robot2Area )
   END_RUNG wire#w4
   RUNG wire#w2
      Contact( "KukaRobot2_CtrlDB".sROBtoPLC.User.Cycle.DO300_HomeInside )
      wire#w5
      Contact( "KukaRobot3_CtrlDB".sROBtoPLC.User.Cycle.DO249_PickMagnetInside )
   END_RUNG wire#w4
   RUNG wire#w5
      Contact( "KukaRobot3_CtrlDB".sROBtoPLC.User.Cycle.DO253_PickGlueNGInside )
   END_RUNG wire#w4
   RUNG wire#w5
      Contact( "KukaRobot3_CtrlDB".sROBtoPLC.User.Cycle.DO281_PressPickInside )
   END_RUNG wire#w4
   RUNG wire#w6
      Contact( "Robot_DB".RobotFlag_3[1] )
      Move(in := 0, out1 => "KukaRobot3_CtrlDB".iSpeedValue)
   END_RUNG
   RUNG wire#w6
      Not()
      Contact( "Robot_DB".RobotFlag_3[1] )
      Contact( "Station_Sys".Auto.Mode )
      { S7_Templates := "time_type := Time" } "Robot_DB".TON[4].TON(pt := T#2S, et =>)
      Move(in := "Robot_DB".RobotSpeed[3], out1 => "KukaRobot3_CtrlDB".iSpeedValue)
      R_Coil( "Robot_DB".RobotFlag_3[1] )
   END_RUNG
   RUNG wire#w1
      I_Contact( "Robot_DB".RobotFlag_3[1] )
      { S7_Templates := "SrcType := USInt" } EQ_Contact(in1 := "KukaRobot3_CtrlDB".iSpeedValue, in2 := 0)
      { S7_Templates := "time_type := Time" } "Robot_DB".TON[7].TON(pt := T#500MS, et =>)
      P_Trig( "Robot_DB".P[13] )
      Move(in := 20, out1 => "KukaRobot3_CtrlDB".iSpeedValue)
   END_RUNG
   RUNG wire#w1
      { S7_Templates := "SrcType := USInt" } GE_Contact(in1 := "KukaRobot3_CtrlDB".iSpeedValue, in2 := 100)
      Move(in := 100, out1 => "KukaRobot3_CtrlDB".iSpeedValue)
   END_RUNG
   RUNG wire#w1
      I_Contact( "Robot_DB".RobotFlag_3[1] )
      I_Contact( "Robot_DB".Robot_3.SpeedChangeFlag )
      I_Contact( "ChangeOver_DB".Global.ScanFixtureFlag )
      Contact( "AlwaysFALSE" )
      Move(in := 20, out1 => "KukaRobot3_CtrlDB".iSpeedValue)
   END_RUNG
   RUNG wire#w1
      Contact( "ChangeOver_DB".Global.ScanFixtureFlag )
      Contact( "AlwaysFALSE" )
      Move(in := 20, out1 => "KukaRobot3_CtrlDB".iSpeedValue)
   END_RUNG
   // the same network as SCL:
   #_w1 := "AlwaysTRUE" AND "Station_Sys".Auto.Mode AND ((NOT "KukaRobot2_CtrlDB".sROBtoPLC.User.Home.DO181_Robot3Area AND ("KukaRobot3_CtrlDB".sROBtoPLC.User.Cycle.DO249_PickMagnetInside OR "KukaRobot3_CtrlDB".sROBtoPLC.User.Cycle.DO253_PickGlueNGInside OR "KukaRobot3_CtrlDB".sROBtoPLC.User.Cycle.DO277_PressPutRingInside OR "KukaRobot3_CtrlDB".sROBtoPLC.User.Cycle.DO281_PressPickInside OR NOT "KukaRobot3_CtrlDB".sROBtoPLC.User.Home.DO178_Robot2Area)) OR ("KukaRobot2_CtrlDB".sROBtoPLC.User.Cycle.DO300_HomeInside AND ("KukaRobot3_CtrlDB".sROBtoPLC.User.Cycle.DO249_PickMagnetInside OR "KukaRobot3_CtrlDB".sROBtoPLC.User.Cycle.DO253_PickGlueNGInside OR "KukaRobot3_CtrlDB".sROBtoPLC.User.Cycle.DO281_PressPickInside))) AND "AlwaysTRUE";
   #_w2 := #_w1 AND NOT "Robot_DB".P[4];   // rising edge
   "Robot_DB".P[4] := #_w1;
   IF #_w2 THEN
       "Robot_DB".RobotSpeed[3] := "KukaRobot3_CtrlDB".sROBtoPLC.User.Public.GO_SpeedActual;
       "Robot_DB".RobotFlag_3[1] := TRUE;
   END_IF;
   IF #_w1 AND "Robot_DB".RobotFlag_3[1] THEN "KukaRobot3_CtrlDB".iSpeedValue := 0; END_IF;
   "Robot_DB".TON[4].TON(IN := NOT #_w1 AND "Robot_DB".RobotFlag_3[1] AND "Station_Sys".Auto.Mode, PT := T#2S);
   IF "Robot_DB".TON[4].Q THEN
       "KukaRobot3_CtrlDB".iSpeedValue := "Robot_DB".RobotSpeed[3];
       "Robot_DB".RobotFlag_3[1] := FALSE;
   END_IF;
   "Robot_DB".TON[7].TON(IN := "AlwaysTRUE" AND NOT "Robot_DB".RobotFlag_3[1] AND ("KukaRobot3_CtrlDB".iSpeedValue = 0),
                         PT := T#500MS);
   #_w3 := "Robot_DB".TON[7].Q AND NOT "Robot_DB".P[13];   // rising edge
   "Robot_DB".P[13] := "Robot_DB".TON[7].Q;
   IF #_w3 THEN "KukaRobot3_CtrlDB".iSpeedValue := 20; END_IF;
   IF "AlwaysTRUE" AND ("KukaRobot3_CtrlDB".iSpeedValue >= 100) THEN
       "KukaRobot3_CtrlDB".iSpeedValue := 100;
   END_IF;
   IF "AlwaysTRUE" AND NOT "Robot_DB".RobotFlag_3[1] AND NOT "Robot_DB".Robot_3.SpeedChangeFlag AND NOT "ChangeOver_DB".Global.ScanFixtureFlag AND "AlwaysFALSE" THEN
       "KukaRobot3_CtrlDB".iSpeedValue := 20;
   END_IF;
   IF "AlwaysTRUE" AND "ChangeOver_DB".Global.ScanFixtureFlag AND "AlwaysFALSE" THEN
       "KukaRobot3_CtrlDB".iSpeedValue := 20;
   END_IF;
END_REGION

REGION Network 37: Robot3 No Task Running
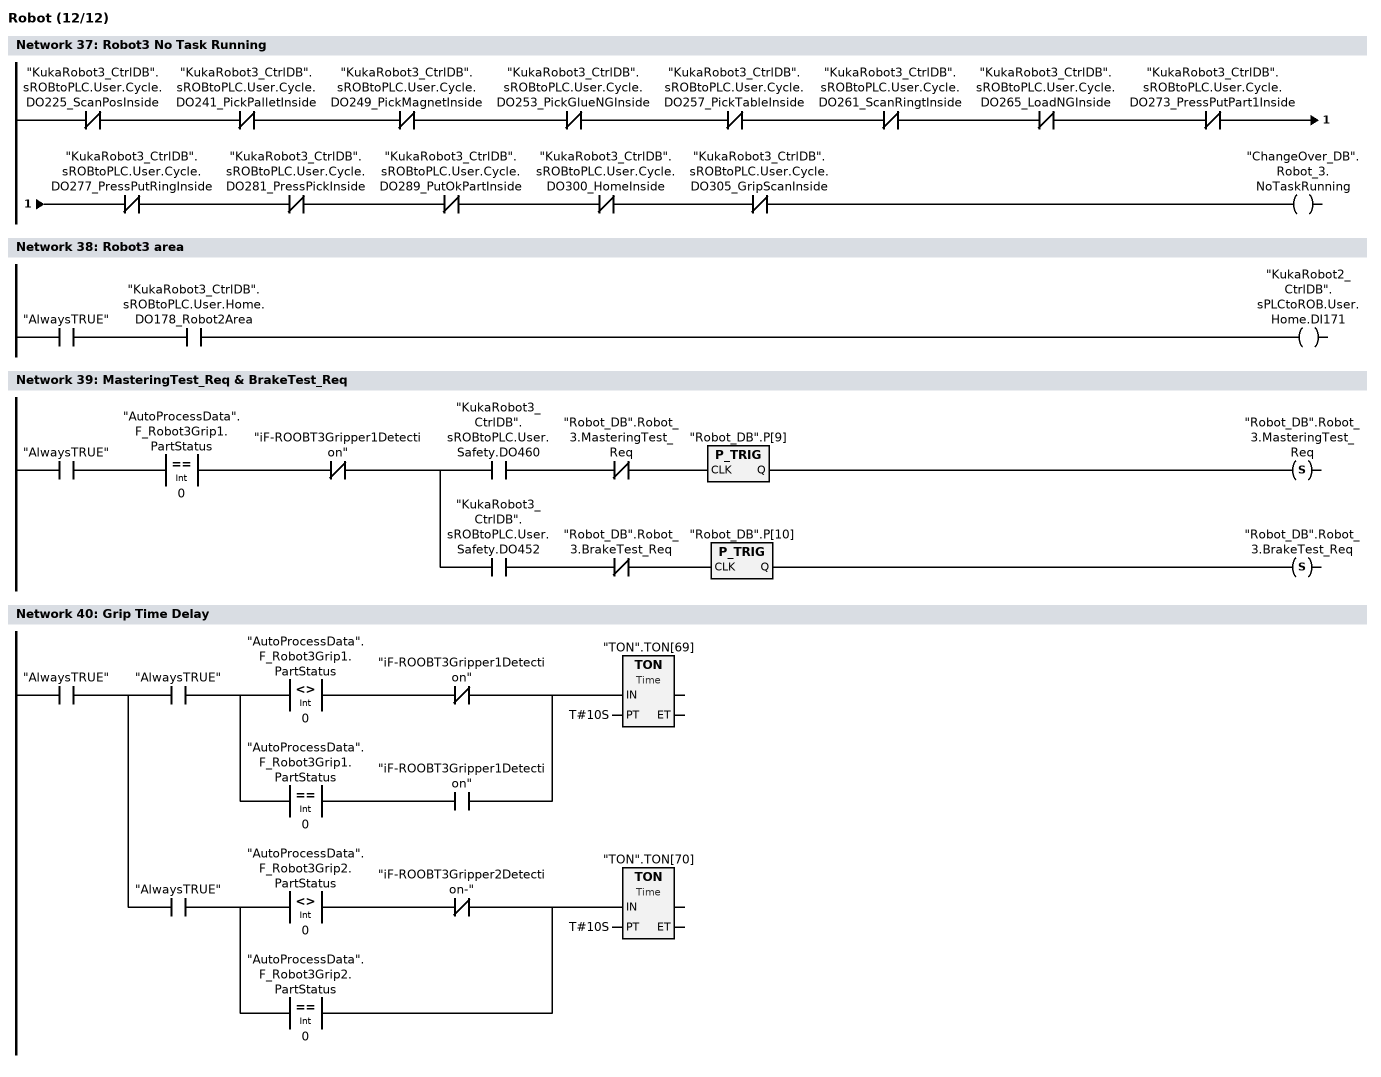
   RUNG wire#powerrail
      I_Contact( "KukaRobot3_CtrlDB".sROBtoPLC.User.Cycle.DO225_ScanPosInside )
      I_Contact( "KukaRobot3_CtrlDB".sROBtoPLC.User.Cycle.DO241_PickPalletInside )
      I_Contact( "KukaRobot3_CtrlDB".sROBtoPLC.User.Cycle.DO249_PickMagnetInside )
      I_Contact( "KukaRobot3_CtrlDB".sROBtoPLC.User.Cycle.DO253_PickGlueNGInside )
      I_Contact( "KukaRobot3_CtrlDB".sROBtoPLC.User.Cycle.DO257_PickTableInside )
      I_Contact( "KukaRobot3_CtrlDB".sROBtoPLC.User.Cycle.DO261_ScanRingtInside )
      I_Contact( "KukaRobot3_CtrlDB".sROBtoPLC.User.Cycle.DO265_LoadNGInside )
      I_Contact( "KukaRobot3_CtrlDB".sROBtoPLC.User.Cycle.DO273_PressPutPart1Inside )
      I_Contact( "KukaRobot3_CtrlDB".sROBtoPLC.User.Cycle.DO277_PressPutRingInside )
      I_Contact( "KukaRobot3_CtrlDB".sROBtoPLC.User.Cycle.DO281_PressPickInside )
      I_Contact( "KukaRobot3_CtrlDB".sROBtoPLC.User.Cycle.DO289_PutOkPartInside )
      I_Contact( "KukaRobot3_CtrlDB".sROBtoPLC.User.Cycle.DO300_HomeInside )
      I_Contact( "KukaRobot3_CtrlDB".sROBtoPLC.User.Cycle.DO305_GripScanInside )
      Coil( "ChangeOver_DB".Robot_3.NoTaskRunning )
   END_RUNG
   // the same network as SCL:
   "ChangeOver_DB".Robot_3.NoTaskRunning := NOT "KukaRobot3_CtrlDB".sROBtoPLC.User.Cycle.DO225_ScanPosInside AND NOT "KukaRobot3_CtrlDB".sROBtoPLC.User.Cycle.DO241_PickPalletInside AND NOT "KukaRobot3_CtrlDB".sROBtoPLC.User.Cycle.DO249_PickMagnetInside AND NOT "KukaRobot3_CtrlDB".sROBtoPLC.User.Cycle.DO253_PickGlueNGInside AND NOT "KukaRobot3_CtrlDB".sROBtoPLC.User.Cycle.DO257_PickTableInside AND NOT "KukaRobot3_CtrlDB".sROBtoPLC.User.Cycle.DO261_ScanRingtInside AND NOT "KukaRobot3_CtrlDB".sROBtoPLC.User.Cycle.DO265_LoadNGInside AND NOT "KukaRobot3_CtrlDB".sROBtoPLC.User.Cycle.DO273_PressPutPart1Inside AND NOT "KukaRobot3_CtrlDB".sROBtoPLC.User.Cycle.DO277_PressPutRingInside AND NOT "KukaRobot3_CtrlDB".sROBtoPLC.User.Cycle.DO281_PressPickInside AND NOT "KukaRobot3_CtrlDB".sROBtoPLC.User.Cycle.DO289_PutOkPartInside AND NOT "KukaRobot3_CtrlDB".sROBtoPLC.User.Cycle.DO300_HomeInside AND NOT "KukaRobot3_CtrlDB".sROBtoPLC.User.Cycle.DO305_GripScanInside;
END_REGION

REGION Network 38: Robot3 area
   RUNG wire#powerrail
      Contact( "AlwaysTRUE" )
      Contact( "KukaRobot3_CtrlDB".sROBtoPLC.User.Home.DO178_Robot2Area )
      Coil( "KukaRobot2_CtrlDB".sPLCtoROB.User.Home.DI171 )
   END_RUNG
   // the same network as SCL:
   "KukaRobot2_CtrlDB".sPLCtoROB.User.Home.DI171 := "AlwaysTRUE" AND "KukaRobot3_CtrlDB".sROBtoPLC.User.Home.DO178_Robot2Area;
END_REGION

REGION Network 39: MasteringTest_Req & BrakeTest_Req
   RUNG wire#powerrail
      Contact( "AlwaysTRUE" )
      { S7_Templates := "SrcType := Int" } EQ_Contact(in1 := "AutoProcessData".F_Robot3Grip1.PartStatus, in2 := 0)
      I_Contact( "iF-ROOBT3Gripper1Detection" )
      wire#w1
      Contact( "KukaRobot3_CtrlDB".sROBtoPLC.User.Safety.DO460 )
      I_Contact( "Robot_DB".Robot_3.MasteringTest_Req )
      P_Trig( "Robot_DB".P[9] )
      S_Coil( "Robot_DB".Robot_3.MasteringTest_Req )
   END_RUNG
   RUNG wire#w1
      Contact( "KukaRobot3_CtrlDB".sROBtoPLC.User.Safety.DO452 )
      I_Contact( "Robot_DB".Robot_3.BrakeTest_Req )
      P_Trig( "Robot_DB".P[10] )
      S_Coil( "Robot_DB".Robot_3.BrakeTest_Req )
   END_RUNG
   // the same network as SCL:
   #_w1 := "AlwaysTRUE" AND ("AutoProcessData".F_Robot3Grip1.PartStatus = 0) AND NOT "iF-ROOBT3Gripper1Detection";
   #_w2 := #_w1 AND "KukaRobot3_CtrlDB".sROBtoPLC.User.Safety.DO460 AND NOT "Robot_DB".Robot_3.MasteringTest_Req;
   #_w3 := #_w2 AND NOT "Robot_DB".P[9];   // rising edge
   "Robot_DB".P[9] := #_w2;
   IF #_w3 THEN "Robot_DB".Robot_3.MasteringTest_Req := TRUE; END_IF;
   #_w4 := #_w1 AND "KukaRobot3_CtrlDB".sROBtoPLC.User.Safety.DO452 AND NOT "Robot_DB".Robot_3.BrakeTest_Req;
   #_w5 := #_w4 AND NOT "Robot_DB".P[10];   // rising edge
   "Robot_DB".P[10] := #_w4;
   IF #_w5 THEN "Robot_DB".Robot_3.BrakeTest_Req := TRUE; END_IF;
END_REGION

REGION Network 40: Grip Time Delay
   RUNG wire#powerrail
      Contact( "AlwaysTRUE" )
      wire#w1
      Contact( "AlwaysTRUE" )
      wire#w2
      { S7_Templates := "SrcType := Int" } NE_Contact(in1 := "AutoProcessData".F_Robot3Grip1.PartStatus, in2 := 0)
      I_Contact( "iF-ROOBT3Gripper1Detection" )
      wire#w3
      { S7_Templates := "time_type := Time" } "TON".TON[69].TON(pt := T#10S, et =>)
   END_RUNG
   RUNG wire#w2
      { S7_Templates := "SrcType := Int" } EQ_Contact(in1 := "AutoProcessData".F_Robot3Grip1.PartStatus, in2 := 0)
      Contact( "iF-ROOBT3Gripper1Detection" )
   END_RUNG wire#w3
   RUNG wire#w1
      Contact( "AlwaysTRUE" )
      wire#w4
      { S7_Templates := "SrcType := Int" } NE_Contact(in1 := "AutoProcessData".F_Robot3Grip2.PartStatus, in2 := 0)
      I_Contact( "iF-ROOBT3Gripper2Detection-" )
      wire#w5
      { S7_Templates := "time_type := Time" } "TON".TON[70].TON(pt := T#10S, et =>)
   END_RUNG
   RUNG wire#w4
      { S7_Templates := "SrcType := Int" } EQ_Contact(in1 := "AutoProcessData".F_Robot3Grip2.PartStatus, in2 := 0)
   END_RUNG wire#w5
   // the same network as SCL:
   "TON".TON[69].TON(IN := "AlwaysTRUE" AND "AlwaysTRUE" AND ((("AutoProcessData".F_Robot3Grip1.PartStatus <> 0) AND NOT "iF-ROOBT3Gripper1Detection") OR (("AutoProcessData".F_Robot3Grip1.PartStatus = 0) AND "iF-ROOBT3Gripper1Detection")),
                     PT := T#10S);
   "TON".TON[70].TON(IN := "AlwaysTRUE" AND "AlwaysTRUE" AND ((("AutoProcessData".F_Robot3Grip2.PartStatus <> 0) AND NOT "iF-ROOBT3Gripper2Detection-") OR ("AutoProcessData".F_Robot3Grip2.PartStatus = 0)),
                     PT := T#10S);
END_REGION
END_FUNCTION
